// TwinCAT 3 PLC project Mediator
// ProgramVersion: 3.1.4022.2
// libraries:
//   Tc2_Standard, * (Beckhoff Automation GmbH)
//   Tc2_System, * (Beckhoff Automation GmbH)
//   Tc2_Utilities, * (Beckhoff Automation GmbH)
//   Tc3_Module, * (Beckhoff Automation GmbH)
//   VisuSymbols,3.5.10.0,System
// project tree:
//   DUTs/ E_DeliveryStatus.TcDUT, E_MediatorReturnCode.TcDUT, E_MessageList.TcDUT, E_PeerReturnCode.TcDUT, E_PeersList.TcDUT, ST_LinkedListUnit.TcDUT, ST_Mailbox.TcDUT, ST_Message.TcDUT, ST_PeerAccount.TcDUT, E_System.TcDUT, ST_TimeStrings.TcDUT
//   / GlobalTextList.TcGTLO, PlcTask.TcTTO, TL_MessageList.TcTLO, TL_PeersList.TcTLO, Visualisierungsmanager.TcVMO (not stored), VISU_TASK.TcTTO
//   POUs/ CONVEYOR_TEST.TcPOU, MEDIATOR_TEST.TcPOU
//   POUs/System/Components/ FB_Sensor.TcPOU
//   POUs/System/ GTL.TcGVL, GVL_Constants.TcGVL, GVL_System.TcGVL, GVL_SystemParams.TcGVL, I_Module.TcIO, I_Sequence.TcIO
//   POUs/System/LinkedList/ FB_GenericLinkedList.TcPOU, FB_MessageLinkedList.TcPOU, FB_PeerLinkedList.TcPOU
//   POUs/System/Logging/ E_LoggingSeverity.TcDUT, FB_Logging.TcPOU
//   POUs/System/Messaging/ FB_Mediator.TcPOU, FB_Peer.TcPOU, I_Peer.TcIO, F_Message.TcPOU
//   POUs/System/Utilities/Concats/ F_Concat10.TcPOU, F_Concat3.TcPOU, F_Concat4.TcPOU, F_Concat5.TcPOU, F_Concat6.TcPOU, F_Concat7.TcPOU, F_Concat8.TcPOU, F_Concat9.TcPOU
//   POUs/System/Utilities/ FB_WhiteSpaces.TcPOU
//   POUs/TestBlocks/Conveyor/ E_ConveyorPeerSequence.TcDUT, FB_Conveyor.TcPOU, FB_Conveyor1Sequence.TcPOU, FB_Conveyor2Sequence.TcPOU, FB_Conveyor3Sequence.TcPOU, FB_Conveyor4Sequence.TcPOU, FB_ConveyorLogSequence.TcPOU, FB_ConveyorPeerSequence.TcPOU, I_ConveyorSequence.TcIO
//   POUs/TestBlocks/ FB_Void.TcPOU
//   Rezeptur/ RecipeManager.TcRMO (not stored)
//   VISUs/Frames/ Frame_Conveyor.TcVIS, Frame_ConveyorGroup.TcVIS, Frame_ConveyorSmallGroup.TcVIS, Frame_Peer.TcVIS
//   VISUs/ VISU_CONVEYOR_TEST.TcVIS, VISU_MEDIATOR_TEST.TcVIS
// real-time tasks:
//   TASK PlcTask: cycle T#10ms, priority 20, ADS port 350
//   TASK VISU_TASK: cycle T#200000us, priority 30, ADS port 351

CONFIGURATION Mediator
    RESOURCE PLC ON TwinCAT3
        TASK PlcTask(INTERVAL := T#10ms, PRIORITY := 20);
        TASK VISU_TASK(INTERVAL := T#200000us, PRIORITY := 30);
        PROGRAM MEDIATOR_TEST WITH PlcTask : MEDIATOR_TEST;
        PROGRAM VISU_PRG WITH VISU_TASK : VISU_PRG;
    END_RESOURCE
END_CONFIGURATION

// ---- DUTs/E_DeliveryStatus.TcDUT
{attribute 'qualified_only'}
{attribute 'strict'}
TYPE E_DeliveryStatus :
(
	eNO_DELIVERY_INFORMATION := 0,
	eDELIVERY_OK,
	eDELIVERY_REJECTED
)UINT;
END_TYPE

// ---- DUTs/E_MediatorReturnCode.TcDUT
//{attribute 'qualified_only'}
//{attribute 'strict'}
TYPE E_MediatorReturnCode :
(
	eNO_RETURN_CODE := 0,
	ePEER_ALREADY_CONNECTED,
	ePEER_CONNECTED,
	eMAX_NUMBER_OF_CONNECTED_PEERS,
	ePEER_NOT_FOUND,
	eMESSAGE_DISPATCHED,
	eMESSAGE_NOT_DISPATCHED,
	eDISPATCHING_MESSAGE
)UINT;
END_TYPE

// ---- DUTs/E_MessageList.TcDUT
//{attribute 'qualified_only'}
//{attribute 'strict'}
TYPE E_MessageList :
(
	eNO_MESSAGE := 1,
	eCONVEYOR_1_AT_TRANSFER_POINT,
	eCONVEYOR_1_RESUMING_OPERATION,
	eCONVEYOR_2_AT_TRANSFER_POINT,
	eCONVEYOR_2_RESUMING_OPERATION,
	eCONVEYOR_3_AT_TRANSFER_POINT,
	eCONVEYOR_3_RESUMING_OPERATION,
	eCONVEYOR_4_AT_TRANSFER_POINT,
	eCONVEYOR_4_RESUMING_OPERATION,
	eCONVEYOR_1_PACKAGE_DELIVERED,
	eCONVEYOR_2_PACKAGE_DELIVERED,
	eCONVEYOR_3_PACKAGE_DELIVERED,
	eCONVEYOR_4_PACKAGE_DELIVERED
)UINT;
END_TYPE

// ---- DUTs/E_PeerReturnCode.TcDUT
{attribute 'qualified_only'}
{attribute 'strict'}
TYPE E_PeerReturnCode :
(
	eNO_RETURN_CODE := 0,
	eMESSAGE_IN_OUTBOX,
	eMAILBOX_BUSY,
	eMAILBOX_EMPTIED,
	eMAILBOX_EMPTY,
	eNO_NEW_MESSAGE,
	eMATCH_FOUND,
	eNO_MATCH_FOUND
)UINT;
END_TYPE

// ---- DUTs/E_PeersList.TcDUT
//{attribute 'qualified_only'}
//{attribute 'strict'}
TYPE E_PeersList :
(
	ePEER_NO_PEER := 1,
	ePEER_CONVEYOR_1,
	ePEER_CONVEYOR_2,
	ePEER_CONVEYOR_3,
	ePEER_CONVEYOR_4
)UINT;
END_TYPE

// ---- DUTs/ST_LinkedListUnit.TcDUT
TYPE ST_LinkedListUnit :
STRUCT
	
	// 		HEAD <--------------  --------------> TAIL
	//				Previous			Next
	
	pNext : POINTER TO ST_LinkedListUnit;
	pPrevious : POINTER TO ST_LinkedListUnit;
	pVoid : POINTER TO PVOID; // Pointer to the data
	
END_STRUCT
END_TYPE

// ---- DUTs/ST_Mailbox.TcDUT
TYPE ST_Mailbox : 
STRUCT
	stInbox : ST_Message;
	stOutbox : ST_Message;
	bNewMessageAvail : BOOL;
	bSendingMessage : BOOL;
	bMessageSent : BOOL;
END_STRUCT
END_TYPE

// ---- DUTs/ST_Message.TcDUT
{attribute 'enable_dynamic_creation'}
TYPE ST_Message :
STRUCT
	eMessage : E_MessageList;
	eFromPeer : E_PeersList;
	eToPeer : E_PeersList;
	eDeliveryStatus : E_DeliveryStatus;
END_STRUCT
END_TYPE

// ---- DUTs/ST_PeerAccount.TcDUT
TYPE ST_PeerAccount :
STRUCT
	iPeer : I_Peer;
	//fbMessagesList : FB_LinkedListCtrl;
	//nodes : ARRAY[1..nMAX_DATA_ELEMENTS] OF T_LinkedListEntry;
	//hList : T_HLINKEDLIST; //linked list handle
	aMessages : ARRAY[1..nMAX_DATA_ELEMENTS] OF ST_Message;
	nStackPointer : UINT := 1;
	rMailbox : REFERENCE TO ST_MAILBOX; 
	bMailboxFull : BOOL;
	bMailboxEmpty : BOOL := TRUE;
	eDispatchRoutineReturnCode : E_MediatorReturnCode;
END_STRUCT
END_TYPE

// ---- DUTs/E_System.TcDUT
TYPE E_System :
(
	NULL := 0
)UINT;
END_TYPE

// ---- DUTs/ST_TimeStrings.TcDUT
TYPE ST_TimeStrings :
STRUCT
	sYear : STRING;
	sMonth : STRING;
	sDayOfWeek : STRING;
	sDay : STRING;
	sHour : STRING;
	sMinute : STRING;
	sSecond : STRING;
	sMilliseconds : STRING;
END_STRUCT
END_TYPE

// ---- POUs/System/Logging/E_LoggingSeverity.TcDUT
TYPE E_LoggingSeverity :
(
	eNO_LOGGING := 0,
	eINFO,
	eWARNING,
	eDEBUG,
	eERROR,
	eALL
);
END_TYPE

// ---- POUs/TestBlocks/Conveyor/E_ConveyorPeerSequence.TcDUT
{attribute 'qualified_only'}
{attribute 'strict'}
TYPE E_ConveyorPeerSequence :
(
	eIDLE := 0,
	eSTOP,
	eSTART,
	eHOME,
	eWAIT_FOR_ACK,
	eSTOP_AT_SIGNAL,
	eRESUME_OPERATION,
	eEND_SEQUENCE
);
END_TYPE

// ---- POUs/System/GTL.TcGVL
{attribute 'qualified_only'}
VAR_GLOBAL
	gtlPeers : ARRAY[1..nAVAILABLE_PEERS] OF STRING;
	gtlMessages : ARRAY[1..nAVAILABLE_MESSAGES] OF STRING;
	gtlDeliveryStatus : ARRAY[1..nAVAILABLE_DELIVERY_STATUSES] OF STRING;
END_VAR

// ---- POUs/System/GVL_Constants.TcGVL
VAR_GLOBAL CONSTANT
	nMAX_DATA_ELEMENTS : UINT := 4;
	nACTUAL_NUM_PEERS : UINT := 4;
	nMAX_PEER_NUMBER : UINT := 100;
	nMAX_LOG_MESSAGES : UINT := 1000;
	nAVAILABLE_MESSAGES : UINT := 13;
	nAVAILABLE_PEERS : UINT := 5;
	nAVAILABLE_DELIVERY_STATUSES : UINT := 5;
END_VAR

// ---- POUs/System/GVL_System.TcGVL
VAR_GLOBAL
	fbLogList : FB_Logging;
END_VAR

// ---- POUs/System/GVL_SystemParams.TcGVL
{attribute 'qualified_only'}
VAR_GLOBAL CONSTANT
	sLogPath : T_MaxString := '\\Vboxsvr\vm_share\LogFile.csv';//'C:\Users\TC-1\Documents\Log\LogFile.csv';
END_VAR

// ---- POUs/System/I_Module.TcIO
INTERFACE I_Module

PROPERTY AccessModuleName : String
GET
END_GET
SET
END_SET
END_PROPERTY

END_INTERFACE

// ---- POUs/System/I_Sequence.TcIO
INTERFACE I_Sequence

END_INTERFACE

// ---- POUs/System/Messaging/I_Peer.TcIO
INTERFACE I_Peer

METHOD M_GetNextMessage : ST_Message
END_METHOD

METHOD M_GetPeerId : E_PeersList
VAR_INPUT
END_VAR
END_METHOD

METHOD M_IsNewMessageAvailable : BOOL
END_METHOD

METHOD M_RetrieveMailbox : REFERENCE TO ST_MAILBOX
VAR_INPUT
END_VAR
END_METHOD

METHOD M_SendMessage : E_PeerReturnCode
VAR_INPUT
	in_stMessage : ST_Message;
END_VAR
END_METHOD

END_INTERFACE

// ---- POUs/TestBlocks/Conveyor/I_ConveyorSequence.TcIO
INTERFACE I_ConveyorSequence EXTENDS I_Sequence

METHOD M_ConveyorSequence : BOOL
VAR_INPUT
	in_rConveyor : REFERENCE TO FB_Conveyor;
END_VAR
END_METHOD

END_INTERFACE

// ---- POUs/MEDIATOR_TEST.TcPOU
PROGRAM MEDIATOR_TEST
VAR
	fbRecipeManCommands : RecipeManCommands;
	aLogUnits : ARRAY[1..nMAX_LOG_MESSAGES] OF ST_LinkedListUnit;
	aLogMessages :  ARRAY[1..nMAX_LOG_MESSAGES] OF T_MaxString;
	i : INT;

	bTest : BOOL;
	bCloseFile : BOOL; 
//--------------------------------------------------------------------------------------------------------------------------------------------
	fbMediator : FB_Mediator;
	aMediatorInitReturnCodes : ARRAY[1..GVL_Constants.nACTUAL_NUM_PEERS] OF BOOL;
	
	aConveyorPeers : ARRAY[1..GVL_Constants.nACTUAL_NUM_PEERS] OF FB_Conveyor;
	aConveyorPeerSequence : ARRAY[1..GVL_Constants.nACTUAL_NUM_PEERS] OF FB_ConveyorPeerSequence;
	
	fbConveyor1Sequence : FB_Conveyor1Sequence;
	fbConveyor2Sequence : FB_Conveyor2Sequence;
	fbConveyor3Sequence : FB_Conveyor3Sequence;
	fbConveyor4Sequence : FB_Conveyor4Sequence;
	
	rConveyor1 : REFERENCE TO FB_Conveyor;
	rConveyor2 : REFERENCE TO FB_Conveyor;
	rConveyor3 : REFERENCE TO FB_Conveyor;
	rConveyor4 : REFERENCE TO FB_Conveyor;
	
	
	{attribute 'OPC.UA.DA' := '1'}
	bInit : BOOL;
	nMainI : UINT;
	
	(*
	//fbCutPeer : FB_Peer(E_PeersList.ePEER_SCHNEIDEN);
	fbDebugPeer1 : FB_Peer(E_PeersList.ePEER_DEBUG_1);
	fbDebugPeer2 : FB_Peer(E_PeersList.ePEER_DEBUG_2);
	
	eMediatorReturnCode : E_MediatorReturnCode;
	
	bPeer1SendMessage : BOOL;
	bPeer2SendMessage : BOOL;
 	*)
	//DEBUG

	
END_VAR


IF bCloseFile THEN
	bCloseFile := FALSE;
	fbLogList.M_CloseFile();
END_IF

fbMediator();
//fbRecipeManCommands();

IF NOT bInit THEN
	
	fbRecipeManCommands.
		LoadAndWriteRecipe(
			RecipeDefinitionName := 'PeersList',
			RecipeName := 'GTL'
		);
		
	fbMediator.AccessModuleName := 'Mediator';
	rConveyor1 REF= aConveyorPeers[1];
	rConveyor1.M_RegisterSequence(fbConveyor1Sequence);
	rConveyor1.AccessModuleName := GTL.gtlPeers[E_PeersList.ePEER_CONVEYOR_1];
	rConveyor2 REF= aConveyorPeers[2];
	rConveyor2.M_RegisterSequence(fbConveyor2Sequence);
	rConveyor3 REF= aConveyorPeers[3];
	rConveyor3.M_RegisterSequence(fbConveyor3Sequence);
	rConveyor4 REF= aConveyorPeers[4];
	rConveyor4.M_RegisterSequence(fbConveyor4Sequence);
	
	rConveyor1.eSetPeerId := E_PeersList.ePEER_CONVEYOR_1;
	rConveyor2.eSetPeerId := E_PeersList.ePEER_CONVEYOR_2;
	rConveyor3.eSetPeerId := E_PeersList.ePEER_CONVEYOR_3; 
	rConveyor4.eSetPeerId := E_PeersList.ePEER_CONVEYOR_4; 
	
	FOR nMainI := 1 TO GVL_Constants.nACTUAL_NUM_PEERS DO 
		aMediatorInitReturnCodes[nMainI] S= 
			(fbMediator.M_AddPeer(aConveyorPeers[nMainI]) = E_MediatorReturnCode.ePEER_CONNECTED);
		//aConveyorPeers[nMainI].M_RegisterSequence(aConveyorPeerSequence[nMainI]);
		aConveyorPeers[nMainI].in_bSystemStart := TRUE;
	END_FOR	
	
	IF 	aMediatorInitReturnCodes[1]  
		AND aMediatorInitReturnCodes[2]
		AND aMediatorInitReturnCodes[3]
		AND aMediatorInitReturnCodes[4]
		THEN
			bInit := TRUE;
	END_IF
ELSE
	
	FOR nMainI := 1 TO GVL_Constants.nACTUAL_NUM_PEERS DO 
		aConveyorPeers[nMainI]();
	END_FOR	
	
END_IF

END_PROGRAM

// ---- POUs/System/Messaging/FB_Mediator.TcPOU
FUNCTION_BLOCK FB_Mediator IMPLEMENTS I_Module

VAR
	aPeersConnected : ARRAY[1..nMAX_PEER_NUMBER] OF ST_PeerAccount;
	aLogMessages :  ARRAY[1..nMAX_LOG_MESSAGES] OF T_MaxString;
	aPeerUnits : ARRAY[1..nMAX_PEER_NUMBER] OF ST_LinkedListUnit;
	aLogUnits : ARRAY[1..nMAX_LOG_MESSAGES] OF ST_LinkedListUnit;
	
	fbPeersList : FB_PeerLinkedList;
	//fbLogList : FB_Logging;
	
	nStackPointer : UINT := 1;
	bAtLeastOnePeerConnected : BOOL;
	bInit : BOOL;
	i : UINT;
	
	stTestUnit : ST_LinkedListUnit;
	pTestMessage : POINTER TO ST_Message;
	stEmptyMessage : ST_MESSAGE;
	sModuleName : STRING;
	
	//DEBUG:
	//If one of the following variables becomes TRUE, investigation of the cause is mandatory
//--------------------------------------------------------------------------------------------
	bFailedToRelocateToTail : BOOL;
	bNullExceptionWhileDispatching : BOOL;
	bNullExceptionWhileCheckingMailbox : BOOL;
//--------------------------------------------------------------------------------------------


END_VAR
VAR CONSTANT
	
END_VAR

M_Init();
M_CheckMailboxes();
M_DispatchMessages();


PROPERTY AccessModuleName : STRING
GET
AccessModuleName := sModuleName;
END_GET
SET
sModuleName := AccessModuleName;
END_SET
END_PROPERTY

METHOD PUBLIC M_AddPeer : E_MediatorReturnCode
VAR_INPUT
	in_iPeer : I_Peer;
END_VAR
VAR
	i : UINT;
	
END_VAR
IF NOT fbPeersList.bInit THEN
	RETURN;
END_IF

IF nStackPointer > nMAX_PEER_NUMBER THEN
	M_AddPeer := E_MediatorReturnCode.eMAX_NUMBER_OF_CONNECTED_PEERS;
	RETURN;
END_IF

FOR i := 1 TO nMAX_PEER_NUMBER DO
	IF aPeersConnected[i].iPeer = in_iPeer THEN
		M_AddPeer := E_MediatorReturnCode.ePEER_ALREADY_CONNECTED;
		RETURN;	
	END_IF
END_FOR

aPeersConnected[nStackPointer].iPeer := in_iPeer;
aPeersConnected[nStackPointer].rMailbox Ref= in_iPeer.M_RetrieveMailbox();

fbPeersList.M_AddPeerToTail
(
	pPeerToAdd := ADR(aPeersConnected[nStackPointer]),
	pUnitToAdd := ADR(aPeerUnits[nStackPointer])
);

nStackPointer := nStackPointer + 1;

bAtLeastOnePeerConnected := TRUE;

M_AddPeer := E_MediatorReturnCode.ePEER_CONNECTED;
END_METHOD

METHOD PRIVATE M_CheckMailboxes : BOOL

VAR
	nSendersAccount : UINT;
	nSendersStackPointer : UINT;
	stMessageToAdd : ST_Message;
	pPeer : POINTER TO ST_PeerAccount;
END_VAR
IF NOT bAtLeastOnePeerConnected THEN
	RETURN;
END_IF 

FOR nSendersAccount := 1 TO nStackPointer-1 DO
	
(*
	IF nSendersAccount = 1 THEN
		fbPeersList.pGetCurrent := fbPeersList.pHead;
		fbPeersList.nGetNextPosition := 1;
	END_IF
*)

	pPeer :=  fbPeersList.M_GetNextPeer();
	
	IF pPeer = NULL THEN
		//Report null exception
		bNullExceptionWhileCheckingMailbox := TRUE;
		CONTINUE;
	END_IF
	
	IF pPeer^.rMailbox.bMessageSent THEN
		pPeer^.rMailbox.bMessageSent := FALSE;
	END_IF;
	
	//If sender has a message in its outbox, add the message to the list of messages
	//The oldest message always in front of the list (FIFO)
	IF pPeer^.rMailbox.bSendingMessage THEN
		
		nSendersStackPointer := pPeer^.nStackPointer;
		// If the senders account has less then X messages, add the outgoing message to the message list 
		IF nSendersStackPointer <= nMAX_DATA_ELEMENTS THEN
	
			stMessageToAdd := pPeer^.rMailbox.stOutbox;
			
			pPeer^.bMailboxFull := FALSE;
			pPeer^.aMessages[nSendersStackPointer] := stMessageToAdd;		
			pPeer^.nStackPointer := nSendersStackPointer + 1;		
			pPeer^.bMailboxEmpty := FALSE;		
			pPeer^.rMailbox.bSendingMessage := FALSE;
			pPeer^.rMailbox.stOutbox := stEmptyMessage;
	
			//Will be true for only one cycle
			pPeer^.rMailbox.bMessageSent := TRUE;
			
		ELSE
			
			//Mailbox contains more than X messages
			pPeer^.bMailboxFull := TRUE;
			
		END_IF
		
	END_IF
	
END_FOR
END_METHOD

METHOD PRIVATE M_DeleteMessageFromSendersAccount : BOOL
VAR_INPUT
	in_pSenderPeer : POINTER TO ST_PeerAccount;
END_VAR
VAR
	stEmptyMessage : ST_MESSAGE;
	nSendersStackPointer : UINT;
	i : UINT;
END_VAR
IF in_pSenderPeer^.bMailboxEmpty THEN
	RETURN;
END_IF 

nSendersStackPointer := in_pSenderPeer^.nStackPointer;
in_pSenderPeer^.nStackPointer := nSendersStackPointer - 1;

//Only one message was in the list
IF in_pSenderPeer^.nStackPointer = 1 THEN
	
	//Remove oldest message from list
	in_pSenderPeer^.aMessages[1] := stEmptyMessage;
	in_pSenderPeer^.bMailboxEmpty := TRUE;
ELSE
	//Move all the messages by one 
	FOR i := 2 TO nSendersStackPointer-1 DO 
		in_pSenderPeer^.aMessages[i - 1] := 
			in_pSenderPeer^.aMessages[i];
	END_FOR
	
	//Remove newest message from list
	in_pSenderPeer^.aMessages[nSendersStackPointer-1] := stEmptyMessage;
	
END_IF
END_METHOD

METHOD PRIVATE M_DispatchMessages 
VAR_INPUT
END_VAR
VAR_OUTPUT
	
END_VAR
VAR
	nSenderPeer : UINT;
	nReceiverPeer : UINT;
	
	pPeer : POINTER TO ST_PeerAccount;
	pUnit : POINTER TO ST_LinkedListUnit;
	
	nPeerListPosition : UINT;
END_VAR

VAR_INST

END_VAR
IF 	NOT bAtLeastOnePeerConnected 
	OR fbPeersList.M_GetCurrentPosition() = 0
	THEN
	
	RETURN;
END_IF 

FOR nSenderPeer := 1 TO nStackPointer-1 DO
(*	
	IF nSenderPeer = 1 THEN
		fbPeersList.pGetCurrent := fbPeersList.pHead;
		fbPeersList.nGetNextPosition := 1;
	END_IF
*)
	pPeer :=  fbPeersList.M_GetNextPeer();
	
	IF pPeer = NULL THEN
		//Report null exception
		bNullExceptionWhileDispatching := TRUE;
		CONTINUE;
	END_IF
	
	//Check if peer has mail to send
	IF NOT pPeer^.bMailboxEmpty THEN
		
		//Result 0 means peer not found
		nReceiverPeer := M_FindPeer( M_GetReceiverPeerId( pPeer ) );
		
		IF nReceiverPeer > 0 THEN
			
			//Sends the message only when the receiver has emptied its own mailbox
			IF 	NOT aPeersConnected[nReceiverPeer].rMailbox.bNewMessageAvail
				THEN				
				
				M_SendMessage
				(
					in_nReceiverPeer := nReceiverPeer,
					in_pSenderPeer := pPeer 
				);
				
				IF pPeer^.aMessages[1].eDeliveryStatus = E_DeliveryStatus.eDELIVERY_REJECTED THEN
					
					fbLogList.M_Info(
						in_iModule:=THIS^,
						in_sMessage:= 
							F_Concat8(
								'Peer ', 
								GTL.gtlPeers[ pPeer^.iPeer.M_GetPeerId() ],
								' sending message back to Peer ',
								GTL.gtlPeers[ M_GetReceiverPeerId( pPeer ) ],
								': ',
								GTL.gtlMessages[ pPeer^.aMessages[1].eMessage ],
								';Delivery status: ',
								GTL.gtlDeliveryStatus[ pPeer^.aMessages[1].eDeliveryStatus ]						
							) 	
					);
					
				ELSE
					
					fbLogList.M_Info(
						in_iModule:=THIS^,
						in_sMessage:= 
							F_Concat8(
								'Peer ', 
								GTL.gtlPeers[ pPeer^.iPeer.M_GetPeerId() ],
								' sending following message to Peer ',
								GTL.gtlPeers[ M_GetReceiverPeerId( pPeer ) ],
								': ',
								GTL.gtlMessages[ pPeer^.aMessages[1].eMessage ],
								';Delivery status: ',
								GTL.gtlDeliveryStatus[ E_DeliveryStatus.eDELIVERY_OK ]						
							) 	
					);
					
				END_IF

				
				M_DeleteMessageFromSendersAccount(in_pSenderPeer := pPeer);	
							
				pPeer^.eDispatchRoutineReturnCode := eMESSAGE_DISPATCHED;
				
				bFailedToRelocateToTail S= NOT fbPeersList.M_RelocateToTail();


			ELSE
				
				pPeer^.eDispatchRoutineReturnCode := eMESSAGE_NOT_DISPATCHED;
				pPeer^.aMessages[1].eDeliveryStatus := E_DeliveryStatus.eRECEIVERS_MAILBOX_NOT_EMPTY;
				
				fbLogList.M_Info(
					in_iModule:=THIS^,
					in_sMessage:= 
						F_Concat8(
							'Peer ', 
							GTL.gtlPeers[ pPeer^.iPeer.M_GetPeerId() ],
							' failed to send following message to Peer ',
							GTL.gtlPeers[ M_GetReceiverPeerId( pPeer ) ],
							': ',
							GTL.gtlMessages[ pPeer^.aMessages[1].eMessage ],
							';Delivery status: ',
							GTL.gtlDeliveryStatus[ pPeer^.aMessages[1].eDeliveryStatus ]						
						) 	
				);	
				
			END_IF
			
		ELSE
			
			// Report peer not found;	
			
			fbLogList.M_Info(
				in_iModule:=THIS^,
				in_sMessage:= 
					F_Concat8(
						'Peer ', 
						GTL.gtlPeers[ pPeer^.iPeer.M_GetPeerId() ],
						' failed to send following message to Peer ',
						GTL.gtlPeers[ M_GetReceiverPeerId( pPeer ) ],
						': ',
						GTL.gtlMessages[ pPeer^.aMessages[1].eMessage ],
						';Delivery status: ',
						GTL.gtlDeliveryStatus[ E_DeliveryStatus.ePEER_NOT_FOUND ]						
					) 	
			);
			M_DeleteMessageFromSendersAccount(in_pSenderPeer := pPeer);	
			pPeer^.eDispatchRoutineReturnCode := ePEER_NOT_FOUND;
			
		END_IF
				
	END_IF
	
END_FOR
END_METHOD

METHOD PRIVATE M_FindPeer : UINT
VAR_INPUT
	in_ePeer : E_PeersList;
END_VAR
VAR
	i : UINT;
END_VAR
IF 	NOT bAtLeastOnePeerConnected 
	OR in_ePeer = NULL 
	THEN
	
	RETURN;
	
END_IF 

//Check if receiver peer is in the peers list and return position of peer in the list
FOR i := 1 TO nStackPointer - 1 DO
	
	IF aPeersConnected[i].iPeer.M_GetPeerId() = in_ePeer THEN
		
		M_FindPeer := i;
		RETURN;
		
	END_IF
	
END_FOR

M_FindPeer := 0;
END_METHOD

METHOD PRIVATE M_GetReceiverPeerId : E_PeersList
VAR_INPUT
	in_pSenderPeer : POINTER TO ST_PeerAccount;
END_VAR
VAR
	pMessage : POINTER TO ST_Message;
END_VAR
//Extract receivers Id from the oldest message in the list
M_GetReceiverPeerId := in_pSenderPeer^.aMessages[1].eToPeer;
END_METHOD

METHOD PRIVATE M_Init : BOOL
VAR_INPUT
END_VAR
fbPeersList.M_InitLinkedList(aPeerUnits);
fbLogList.M_InitLinkedList(aLogUnits);
fbLogList(in_sPath := GVL_SystemParams.sLogPath);

IF NOT bInit THEN
	bInit := TRUE;
	
	fbLogList.AccessLoggingSeverity := eALL;
	
	FOR i := 1 TO nMAX_LOG_MESSAGES DO
		aLogUnits[i].pVoid := ADR(aLogMessages[i]);
		fbLogList.M_AddToTail(ADR(aLogUnits[i]));
	END_FOR

END_IF
END_METHOD

METHOD PUBLIC M_IsPeerConnected : BOOL
VAR_INPUT
	in_ePeer : E_PeersList;
END_VAR
VAR
	i : UINT;
END_VAR
FOR i := 1 TO nMAX_PEER_NUMBER DO
	
	IF aPeersConnected[i].iPeer.M_GetPeerId() = in_ePeer THEN
		
		M_IsPeerConnected := TRUE;
		RETURN;
		
	END_IF
	
END_FOR
END_METHOD

METHOD PRIVATE M_SendMessage : BOOL
VAR_INPUT
	in_nReceiverPeer : UINT;
	in_pSenderPeer : POINTER TO ST_PeerAccount;
END_VAR
//Dispatch mail after the FIFO principle
aPeersConnected[in_nReceiverPeer].rMailbox.stInbox := in_pSenderPeer^.aMessages[1];
aPeersConnected[in_nReceiverPeer].rMailbox.bNewMessageAvail := TRUE;
END_METHOD

END_FUNCTION_BLOCK

// ---- POUs/System/LinkedList/FB_PeerLinkedList.TcPOU
FUNCTION_BLOCK FB_PeerLinkedList EXTENDS FB_GenericLinkedList
VAR_INPUT
END_VAR
VAR_OUTPUT
END_VAR
VAR
END_VAR

METHOD M_AddPeerToHead : BOOL
VAR_INPUT
	pUnitToAdd : POINTER TO ST_LinkedListUnit;
	pPeerToAdd : POINTER TO ST_PeerAccount;
END_VAR
pUnitToAdd^.pVoid := pPeerToAdd;
SUPER^.M_AddToHead(pUnitToAdd);
END_METHOD

METHOD M_AddPeerToTail : BOOL
VAR_INPUT
	pUnitToAdd : POINTER TO ST_LinkedListUnit;
	pPeerToAdd : POINTER TO ST_PeerAccount;
END_VAR
pUnitToAdd^.pVoid := pPeerToAdd;
SUPER^.M_AddToTail(pUnitToAdd);
END_METHOD

METHOD M_GetHeadPeer : POINTER TO ST_PeerAccount
VAR_INPUT
END_VAR
VAR
	stUnit : POINTER TO ST_LinkedListUnit;
END_VAR
stUnit := SUPER^.M_GetHead();

IF stUnit = NULL THEN
	RETURN;
END_IF

M_GetHeadPeer := stUnit^.pVoid;
END_METHOD

METHOD M_GetNextPeer : POINTER TO ST_PeerAccount
VAR_INPUT
END_VAR
VAR
	stUnit : POINTER TO ST_LinkedListUnit;
END_VAR
stUnit := SUPER^.M_GetNext();

IF stUnit = NULL THEN
	RETURN;
END_IF

M_GetNextPeer := stUnit^.pVoid;
END_METHOD

METHOD M_GetTailPeer : POINTER TO ST_PeerAccount
VAR_INPUT
END_VAR
VAR
	stUnit : POINTER TO ST_LinkedListUnit;
END_VAR
stUnit := SUPER^.M_GetTail();

IF stUnit = NULL THEN
	RETURN;
END_IF

M_GetTailPeer := stUnit^.pVoid;
END_METHOD

END_FUNCTION_BLOCK

// ---- POUs/System/LinkedList/FB_GenericLinkedList.TcPOU
FUNCTION_BLOCK FB_GenericLinkedList
VAR_INPUT
END_VAR
VAR_OUTPUT
	bInit : BOOL;
END_VAR
VAR
	
	pHead : POINTER TO ST_LinkedListUnit;
	pTail : POINTER TO ST_LinkedListUnit;
	pPointer : POINTER TO ST_LinkedListUnit; //Helper
	
	//pGetNext : POINTER TO ST_LinkedListUnit;
	nGetNextPosition : UINT := 1;
	
	pGetCurrent : POINTER TO ST_LinkedListUnit;
	nGetCurrentPosition : UINT := 1;
	
	nSizeOfLinkedList : DINT;
	
	bIsEmpty : BOOL := TRUE;
	bIsFull : BOOL;
	nUnitsInTheList : DINT;
	
		//DEBUG:
	//If one of the following variables becomes TRUE, investigation of the cause is mandatory
//--------------------------------------------------------------------------------------------
	bTriedToRelocatePositionZero : BOOL;
//--------------------------------------------------------------------------------------------
END_VAR

METHOD M_AddToHead : BOOL
VAR_INPUT
	pUnitToAdd : POINTER TO ST_LinkedListUnit;
END_VAR
IF bIsFull THEN
	RETURN;
END_IF

IF bIsEmpty THEN
	pHead := pUnitToAdd;
	pGetCurrent := pHead;
	pTail := pHead;
	pPointer := pHead;
ELSE
	pHead^.pPrevious := pUnitToAdd;
	pUnitToAdd^.pNext := pHead;
	pUnitToAdd^.pPrevious := NULL;
	pHead := pUnitToAdd;	
END_IF

nUnitsInTheList := nUnitsInTheList + 1;
M_CheckUnitsInTheList();

M_AddToHead := TRUE;
END_METHOD

METHOD M_AddToTail : BOOL
VAR_INPUT
	pUnitToAdd : POINTER TO ST_LinkedListUnit;
END_VAR
IF bIsFull THEN
	RETURN;
END_IF

IF bIsEmpty THEN
	pHead := pUnitToAdd;
	pGetCurrent := pHead;
	pTail := pHead;
	pPointer := pHead;
ELSE
	pTail^.pNext := pUnitToAdd;
	pUnitToAdd^.pPrevious := pTail;
	pUnitToAdd^.pNext := NULL;
	pTail := pUnitToAdd;	
END_IF

nUnitsInTheList := nUnitsInTheList + 1;
M_CheckUnitsInTheList();
	
M_AddToTail := TRUE;
END_METHOD

METHOD M_CheckUnitsInTheList : BOOL
VAR_INPUT
END_VAR
IF nUnitsInTheList = nSizeOfLinkedList THEN
	bIsFull := TRUE;
ELSIF nUnitsInTheList < nSizeOfLinkedList THEN
	bIsFull := FALSE;
END_IF

IF nUnitsInTheList > 0 THEN
	bIsEmpty := FALSE;
ELSIF nUnitsInTheList = 0 THEN
	bIsEmpty := TRUE;
END_IF
END_METHOD

METHOD M_FindUnit : BOOL
VAR_INPUT
END_VAR
END_METHOD

METHOD M_GetCurrent : POINTER TO ST_LinkedListUnit
VAR_INPUT
END_VAR
IF bIsEmpty THEN
	RETURN;
END_IF

M_GetCurrent := pGetCurrent;
END_METHOD

METHOD M_GetCurrentPosition : UINT
VAR_INPUT
END_VAR
M_GetCurrentPosition := nGetCurrentPosition;
END_METHOD

METHOD M_GetHead : POINTER TO ST_LinkedListUnit
IF bIsEmpty THEN
	RETURN;
END_IF

M_GetHead := pHead;
END_METHOD

//Gets the next Unit and moves the current pointer forward
METHOD M_GetNext : POINTER TO ST_LinkedListUnit
IF bIsEmpty THEN
	RETURN;
END_IF

//If the search pointer reaches the end, reset the counter and the pointer
IF pGetCurrent = NULL THEN
	pGetCurrent := pHead;
	nGetNextPosition := 1;
	M_GetNext := pGetCurrent;
	//pGetCurrent := pGetCurrent^.pNext;
ELSE
	M_GetNext := pGetCurrent;
	//pGetCurrent := pGetCurrent^.pNext;
END_IF
pGetCurrent := pGetCurrent^.pNext;
nGetCurrentPosition := nGetNextPosition;
//IF nGetCurrentPosition = nUnitsInTheList THEN
//	nGetNextPosition := 1;
//ELSE
	nGetNextPosition := nGetNextPosition + 1;
//END_IF
END_METHOD

METHOD M_GetTail : POINTER TO ST_LinkedListUnit
IF bIsEmpty THEN
	RETURN;
END_IF

M_GetTail := pTail;
END_METHOD

METHOD M_InitLinkedList : BOOL
VAR_IN_OUT
    aLinkedListMemory : ARRAY [*] OF ST_LinkedListUnit;
END_VAR
VAR
	i : DINT;
	nLowerBound : DINT;
	nUpperBound : DINT;
END_VAR
IF bInit THEN
	RETURN;
END_IF

nLowerBound := LOWER_BOUND(aLinkedListMemory,1);
nUpperBound := UPPER_BOUND(aLinkedListMemory,1);

nSizeOfLinkedList := (nUpperBound - nLowerBound) + 1;


bIsEmpty := TRUE;
bInit := TRUE;
M_InitLinkedList := TRUE;
END_METHOD

METHOD M_RelocateHeadToTail : BOOL
VAR
	pUnit : POINTER TO ST_LinkedListUnit;
END_VAR
pUnit := M_RemoveAtLocation(1);

IF pUnit = NULL THEN
	RETURN;
END_IF

//If the current element is the head
//reset counters
(*
IF pUnit = pGetCurrent THEN
	pGetCurrent := pGetCurrent^.pNext;
	nGetNextPosition := 2;
	nGetCurrentPosition := 1;
END_IF
*)
IF M_AddToTail(pUnit) THEN
	M_RelocateHeadToTail := TRUE;
END_IF
END_METHOD

METHOD M_RelocateToHead : BOOL
VAR
	pUnit : POINTER TO ST_LinkedListUnit;
END_VAR
pUnit := M_RemoveAtLocation(M_GetCurrentPosition());

IF pUnit = NULL THEN
	RETURN;
END_IF

IF M_AddToHead(pUnit) THEN
	M_RelocateToHead := TRUE;
END_IF
END_METHOD

METHOD M_RelocateToTail : BOOL
VAR_INPUT
END_VAR
VAR
	pUnit : POINTER TO ST_LinkedListUnit;
END_VAR
pUnit := M_RemoveAtLocation(M_GetCurrentPosition());

IF pUnit = NULL THEN
	RETURN;
END_IF

IF M_AddToTail(pUnit) THEN
	M_RelocateToTail := TRUE;
END_IF
END_METHOD

METHOD M_RemoveAtLocation : POINTER TO ST_LinkedListUnit
VAR_INPUT
	in_nLocation : UINT;
END_VAR
VAR
	nCounter : UINT;
END_VAR
IF 	bIsEmpty 
	OR in_nLocation > nUnitsInTheList
	OR in_nLocation = 0
	THEN
	
	IF  in_nLocation = 0 
		AND NOT bIsEmpty 
		THEN
		
		bTriedToRelocatePositionZero := TRUE;
	END_IF
	
	RETURN;
END_IF

pPointer := pHead;
IF in_nLocation = 1 THEN
	M_RemoveAtLocation := M_RemoveHead();
	RETURN;
ELSIF in_nLocation = nUnitsInTheList THEN
	M_RemoveAtLocation := M_RemoveTail();
	RETURN;
ELSE
	
	FOR nCounter := 2 TO in_nLocation DO
		pPointer := pPointer^.pNext;
	END_FOR

END_IF

M_RemoveAtLocation := pPointer;

nUnitsInTheList := nUnitsInTheList - 1;
M_CheckUnitsInTheList();

pPointer := pPointer^.pPrevious;
pPointer^.pNext := pPointer^.pNext^.pNext;
pPointer := pPointer^.pNext;
pPointer^.pPrevious := pPointer^.pPrevious^.pPrevious;
END_METHOD

METHOD M_RemoveHead : POINTER TO ST_LinkedListUnit
VAR_INPUT
END_VAR
IF bIsEmpty THEN
	RETURN;
END_IF

M_RemoveHead := pHead;

IF nUnitsInTheList = 1 THEN
	nUnitsInTheList := 0;
	bIsEmpty := TRUE;	
	pHead := NULL;
	pTail := NULL;
	pPointer := NULL;
ELSE
	pHead := pHead^.pNext;
	pHead^.pPrevious := NULL; 	
	nUnitsInTheList := nUnitsInTheList - 1;
END_IF

M_CheckUnitsInTheList();
END_METHOD

METHOD M_RemoveTail : POINTER TO ST_LinkedListUnit
VAR_INPUT
END_VAR
IF bIsEmpty THEN
	RETURN;
END_IF

M_RemoveTail := pTail;

IF nUnitsInTheList = 1 THEN
	nUnitsInTheList := 0;
	bIsEmpty := TRUE;	
	pHead := NULL;
	pTail := NULL;
	pPointer := NULL;
ELSE
	pTail := pTail^.pPrevious;
	pTail^.pNext := NULL; 	
	nUnitsInTheList := nUnitsInTheList - 1;
END_IF

M_CheckUnitsInTheList();
END_METHOD

END_FUNCTION_BLOCK

// ---- POUs/System/Utilities/Concats/F_Concat8.TcPOU
FUNCTION F_Concat8 : STRING(255)
VAR_INPUT
	String1 : STRING(255);
	String2 : STRING(255);
	String3 : STRING(255);
	String4 : STRING(255);
	String5 : STRING(255);
	String6 : STRING(255);
	String7 : STRING(255);
	String8 : STRING(255);
END_VAR
VAR
END_VAR

F_Concat8 := F_Concat7(String2,String3,String4,String5,String6,String7,String8);
F_Concat8 := CONCAT(String1,F_Concat8);

END_FUNCTION

// ---- POUs/System/Utilities/Concats/F_Concat7.TcPOU
FUNCTION F_Concat7 : STRING(255)
VAR_INPUT
	String1 : STRING(255);
	String2 : STRING(255);
	String3 : STRING(255);
	String4 : STRING(255);
	String5 : STRING(255);
	String6 : STRING(255);
	String7 : STRING(255);
END_VAR
VAR
END_VAR

F_Concat7 := F_Concat6(String2,String3,String4,String5,String6,String7);
F_Concat7 := CONCAT(String1,F_Concat7);

END_FUNCTION

// ---- POUs/System/Utilities/Concats/F_Concat6.TcPOU
FUNCTION F_Concat6 : STRING(255)
VAR_INPUT
	String1 : STRING(255);
	String2 : STRING(255);
	String3 : STRING(255);
	String4 : STRING(255);
	String5 : STRING(255);
	String6 : STRING(255);
END_VAR
VAR
END_VAR

F_Concat6 := F_Concat5(String2,String3,String4,String5,String6);
F_Concat6 := CONCAT(String1,F_Concat6);

END_FUNCTION

// ---- POUs/System/Utilities/Concats/F_Concat5.TcPOU
FUNCTION F_Concat5 : STRING(255)
VAR_INPUT
	String1 : STRING(255);
	String2 : STRING(255);
	String3 : STRING(255);
	String4 : STRING(255);
	String5 : STRING(255);
END_VAR
VAR
END_VAR

F_Concat5 := F_Concat4(String2,String3,String4,String5);
F_Concat5 := CONCAT(String1,F_Concat5);

END_FUNCTION

// ---- POUs/System/Utilities/Concats/F_Concat4.TcPOU
FUNCTION F_Concat4 : STRING(255)
VAR_INPUT
	String1 : STRING(255);
	String2 : STRING(255);
	String3 : STRING(255);
	String4 : STRING(255);
END_VAR
VAR
END_VAR

F_Concat4 := F_CONCAT3(String2,String3,String4);
F_Concat4 := CONCAT(String1,F_Concat4);

END_FUNCTION

// ---- POUs/System/Utilities/Concats/F_Concat3.TcPOU
FUNCTION F_Concat3 : STRING(255)
VAR_INPUT
	String1 : STRING(255);
	String2 : STRING(255);
	String3 : STRING(255);
END_VAR
VAR
END_VAR

F_Concat3 := CONCAT(String1,CONCAT(String2,String3));

END_FUNCTION

// ---- POUs/TestBlocks/Conveyor/FB_Conveyor.TcPOU
FUNCTION_BLOCK FB_Conveyor EXTENDS FB_Peer IMPLEMENTS I_Module
VAR_INPUT
	in_bSystemStart : BOOL;
	in_bStop : BOOL;
	in_bStart : BOOL;
END_VAR
VAR_OUTPUT
	out_fbSensorStop : FB_Sensor;
	out_fbSensorMaterialDispatch : FB_Sensor;
	out_fbSensorSignal : FB_Sensor;
END_VAR
VAR	
	{attribute 'OPC.UA.DA' := '1'}
	bStartMotor AT%Q* : BOOL;
	iSequence : I_ConveyorSequence;
	sModuleName : STRING;
END_VAR

M_CallComponents();
IF in_bSystemStart THEN
	M_RunSequence();
END_IF

PROPERTY AccessModuleName : STRING
GET
AccessModuleName := sModuleName;
END_GET
SET
sModuleName := AccessModuleName;
END_SET
END_PROPERTY

METHOD M_CallComponents : E_PeerReturnCode
VAR_INPUT
END_VAR
out_fbSensorSignal();
out_fbSensorMaterialDispatch();
out_fbSensorStop();
END_METHOD

METHOD M_RegisterSequence : BOOL
VAR_INPUT
	in_iSequence : I_ConveyorSequence;
END_VAR
iSequence := in_iSequence;
END_METHOD

METHOD M_RunSequence : BOOL
VAR_INPUT
END_VAR
IF iSequence = NULL THEN
	RETURN;
END_IF

iSequence.M_ConveyorSequence(this^);
END_METHOD

METHOD M_StartConveyor : BOOL
VAR_INPUT
END_VAR
bStartMotor := TRUE;
END_METHOD

METHOD M_StopConveyor : E_PeerReturnCode
VAR_INPUT
END_VAR
bStartMotor := FALSE;
END_METHOD

END_FUNCTION_BLOCK

// ---- POUs/System/Messaging/FB_Peer.TcPOU
FUNCTION_BLOCK FB_Peer IMPLEMENTS I_Peer
VAR_INPUT
END_VAR
VAR_OUTPUT
END_VAR
VAR
	ePeer : E_PeersList;
	stMailbox : ST_Mailbox; 
END_VAR

PROPERTY eSetPeerId : E_PeersList
SET
ePeer := eSetPeerId;
END_SET
END_PROPERTY

METHOD M_CompareMessage : E_PeerReturnCode
VAR_INPUT
	in_stMessage : ST_Message;
END_VAR
VAR
	stIncomingMessage : ST_MESSAGE;
END_VAR
IF M_IsNewMessageAvailable() THEN
	
	stIncomingMessage := M_GetNextMessage();
	IF 	stIncomingMessage.eMessage = in_stMessage.eMessage
		AND stIncomingMessage.eFromPeer = in_stMessage.eFromPeer
		THEN
		
		M_CompareMessage := E_PeerReturnCode.eMATCH_FOUND;
		
	ELSE
		
		M_CompareMessage := E_PeerReturnCode.eNO_MATCH_FOUND;
	
	END_IF
	
ELSE

	M_CompareMessage := E_PeerReturnCode.eNO_NEW_MESSAGE;	
	
END_IF
END_METHOD

METHOD M_CompareMessageAndEmptyMailbox : E_PeerReturnCode
VAR_INPUT
	in_stMessage : ST_Message;
END_VAR
VAR
	stMessage : ST_Message;
	eTmpEval : E_PeerReturnCode;
END_VAR
M_CompareMessageAndEmptyMailbox := M_CompareMessage(in_stMessage);

IF M_CompareMessageAndEmptyMailbox = E_PeerReturnCode.eNO_MATCH_FOUND THEN
	stMessage := M_GetNextMessage();
	stMessage.eDeliveryStatus := E_DeliveryStatus.eDELIVERY_REJECTED;
	stMessage.eToPeer := stMessage.eFromPeer;
	stMessage.eFromPeer := M_GetPeerId();
	eTmpEval := M_SendMessage(stMessage);
END_IF

IF eTmpEval = E_PeerReturnCode.eMESSAGE_IN_OUTBOX
	OR M_CompareMessageAndEmptyMailbox = E_PeerReturnCode.eMATCH_FOUND
	THEN
	
	M_EmptyMailbox();
	
END_IF
END_METHOD

METHOD M_EmptyMailbox : E_PeerReturnCode
VAR_INPUT
END_VAR
VAR
	stEmptyMessage : ST_MESSAGE;
END_VAR
IF M_IsNewMessageAvailable() THEN
	stMailbox.stInbox := stEmptyMessage;
	stMailbox.bNewMessageAvail := FALSE;
	M_EmptyMailbox := E_PeerReturnCode.eMAILBOX_EMPTIED;
ELSE
	M_EmptyMailbox := E_PeerReturnCode.eMAILBOX_EMPTY;
END_IF
END_METHOD

METHOD M_GetNextMessage : ST_Message
IF M_IsNewMessageAvailable() THEN
	M_GetNextMessage := stMailbox.stInbox;
END_IF
END_METHOD

METHOD M_GetPeerId : E_PeersList
M_GetPeerId := ePeer;
END_METHOD

METHOD M_IsNewMessageAvailable : BOOL
M_IsNewMessageAvailable := stMailbox.bNewMessageAvail;
END_METHOD

METHOD M_RetrieveMailbox : REFERENCE TO ST_MAILBOX
VAR_INPUT
END_VAR
M_RetrieveMailbox Ref= stMailbox;
END_METHOD

METHOD M_SendMessage : E_PeerReturnCode
VAR_INPUT
	in_stMessage : ST_Message;
END_VAR
IF NOT stMailbox.bSendingMessage THEN
	stMailbox.stOutbox := in_stMessage;
	stMailbox.bSendingMessage := TRUE;
	M_SendMessage := E_PeerReturnCode.eMESSAGE_IN_OUTBOX;
ELSE
	M_SendMessage := E_PeerReturnCode.eMAILBOX_BUSY;
END_IF
END_METHOD

END_FUNCTION_BLOCK

// ---- POUs/System/Components/FB_Sensor.TcPOU
FUNCTION_BLOCK FB_Sensor
VAR_INPUT
END_VAR
VAR_OUTPUT
END_VAR
VAR
	{attribute 'OPC.UA.DA' := '1'}
	bSignal  AT%I* : BOOL;	
	fbRTrig : R_TRIG;
END_VAR

fbRTrig(CLK:= bSignal, Q=> );

PROPERTY GetSignal : BOOL
GET
GetSignal := bSignal;
END_GET
END_PROPERTY

PROPERTY GetTriggerSignal : BOOL
GET
GetTriggerSignal := fbRTrig.Q;
END_GET
END_PROPERTY

END_FUNCTION_BLOCK

// ---- POUs/TestBlocks/Conveyor/FB_ConveyorPeerSequence.TcPOU
FUNCTION_BLOCK FB_ConveyorPeerSequence IMPLEMENTS I_ConveyorSequence
VAR_INPUT

END_VAR
VAR_OUTPUT
END_VAR
VAR
	nStep : E_ConveyorPeerSequence;
END_VAR

METHOD M_ConveyorAction : BOOL
VAR_INPUT
	in_stFirstMessage : ST_Message;
	in_stMessageToWaitFor : ST_Message;
	in_stSecondMessage : ST_Message;
	in_rConveyor : REFERENCE TO FB_Conveyor;
END_VAR
VAR_INST
	nConveyorActionStep : UINT;
END_VAR
CASE nConveyorActionStep OF
	
	0:
		IF 	in_rConveyor.M_SendMessage
			(	
				in_stFirstMessage
			) 
			= E_PeerReturnCode.eMESSAGE_IN_OUTBOX 
			THEN
			
			nConveyorActionStep := 10;
			
		END_IF
		
	10:
		
	
		IF 	in_rConveyor.M_CompareMessageAndEmptyMailbox
			(	
				in_stMessageToWaitFor
			) 
			= E_PeerReturnCode.eMATCH_FOUND 
			THEN
			
			nConveyorActionStep := 20;
			
		END_IF

	20:
		
		IF 	in_rConveyor.M_SendMessage
			(	
				in_stSecondMessage
			) 
			= E_PeerReturnCode.eMESSAGE_IN_OUTBOX 
			THEN
			
			nConveyorActionStep := 0;
			M_ConveyorAction := TRUE;
			
		END_IF
		
END_CASE
END_METHOD


METHOD M_ConveyorSequence : BOOL
VAR_INPUT
	in_rConveyor : REFERENCE TO FB_Conveyor;
END_VAR
CASE nStep OF
	
	E_ConveyorPeerSequence.eIDLE:
	
		IF in_rConveyor.in_bStart THEN
			nStep := E_ConveyorPeerSequence.eSTART;
		END_IF
				
	E_ConveyorPeerSequence.eSTART:
		
		in_rConveyor.M_StartConveyor();
		nStep := E_ConveyorPeerSequence.eSTOP_AT_SIGNAL;

	E_ConveyorPeerSequence.eSTOP_AT_SIGNAL:
	
		IF in_rConveyor.out_fbSensorStop.GetTriggerSignal THEN
			in_rConveyor.M_StopConveyor();
			nStep := E_ConveyorPeerSequence.eWAIT_FOR_ACK;
		END_IF
	
	E_ConveyorPeerSequence.eWAIT_FOR_ACK:
		
		IF M_SubjectiveAction(in_rConveyor) THEN
			nStep := E_ConveyorPeerSequence.eRESUME_OPERATION;
		END_IF
	
	E_ConveyorPeerSequence.eRESUME_OPERATION:
		
		in_rConveyor.M_StartConveyor();
		IF in_rConveyor.out_fbSensorMaterialDispatch.GetTriggerSignal THEN
			in_rConveyor.M_StopConveyor();
			nStep := E_ConveyorPeerSequence.eEND_SEQUENCE;
		END_IF
	
	E_ConveyorPeerSequence.eEND_SEQUENCE:
		
END_CASE
END_METHOD

METHOD M_SubjectiveAction : BOOL
VAR_INPUT
	in_rConveyor : REFERENCE TO FB_Conveyor;
END_VAR

VAR
	stFirstMessageToSend : ST_Message;
	stMessageToWaitFor : ST_Message;
	stSecondMessageToSend : ST_Message;
END_VAR
CASE in_rConveyor.M_GetPeerId() OF

	E_PeersList.ePEER_CONVEYOR_1:
	
		stFirstMessageToSend :=
			F_Message(
				eFromPeer := ePEER_CONVEYOR_1,
				eToPeer := ePEER_CONVEYOR_2,
				eMessage := eCONVEYOR_1_AT_TRANSFER_POINT
			);
			
		stMessageToWaitFor := 
			F_Message(
				eFromPeer := ePEER_CONVEYOR_4,
				eToPeer := ePEER_CONVEYOR_1,
				eMessage := eCONVEYOR_4_AT_TRANSFER_POINT
			);
			
		stSecondMessageToSend := 
			F_Message(
				eFromPeer := ePEER_CONVEYOR_1,
				eToPeer := ePEER_CONVEYOR_2,
				eMessage := eCONVEYOR_1_RESUMING_OPERATION
			);
			
	E_PeersList.ePEER_CONVEYOR_2:
		
		stFirstMessageToSend :=
			F_Message(
				eFromPeer := ePEER_CONVEYOR_2,
				eToPeer := ePEER_CONVEYOR_3,
				eMessage := eCONVEYOR_2_AT_TRANSFER_POINT
			);
			
		stMessageToWaitFor := 
			F_Message(
				eFromPeer := ePEER_CONVEYOR_1,
				eToPeer := ePEER_CONVEYOR_2,
				eMessage := eCONVEYOR_1_RESUMING_OPERATION
			);
			
		stSecondMessageToSend := 
			F_Message(
				eFromPeer := ePEER_CONVEYOR_2,
				eToPeer := ePEER_CONVEYOR_3,
				eMessage := eCONVEYOR_2_RESUMING_OPERATION
			);	
	
	E_PeersList.ePEER_CONVEYOR_3:
	
		stFirstMessageToSend :=
			F_Message(
				eFromPeer := ePEER_CONVEYOR_3,
				eToPeer := ePEER_CONVEYOR_4,
				eMessage := eCONVEYOR_3_AT_TRANSFER_POINT
			);
			
		stMessageToWaitFor := 
			F_Message(
				eFromPeer := ePEER_CONVEYOR_2,
				eToPeer := ePEER_CONVEYOR_3,
				eMessage := eCONVEYOR_2_RESUMING_OPERATION
			);
			
		stSecondMessageToSend := 
			F_Message(
				eFromPeer := ePEER_CONVEYOR_3,
				eToPeer := ePEER_CONVEYOR_4,
				eMessage := eCONVEYOR_3_RESUMING_OPERATION
			);
	
	E_PeersList.ePEER_CONVEYOR_4:
	
		stFirstMessageToSend :=
			F_Message(
				eFromPeer := ePEER_CONVEYOR_4,
				eToPeer := ePEER_CONVEYOR_1,
				eMessage := eCONVEYOR_4_AT_TRANSFER_POINT
			);
			
		stMessageToWaitFor := 
			F_Message(
				eFromPeer := ePEER_CONVEYOR_3,
				eToPeer := ePEER_CONVEYOR_4,
				eMessage := eCONVEYOR_3_RESUMING_OPERATION
			);
			
		stSecondMessageToSend := 
			F_Message(
				eFromPeer := ePEER_CONVEYOR_4,
				eToPeer := ePEER_NO_PEER,
				eMessage := eNO_MESSAGE
			);	

END_CASE

M_SubjectiveAction := 
	M_ConveyorAction(
		in_rConveyor := in_rConveyor,
		in_stFirstMessage := stFirstMessageToSend,
		in_stMessageToWaitFor := stMessageToWaitFor,
		in_stSecondMessage := stSecondMessageToSend
	);
END_METHOD

END_FUNCTION_BLOCK

// ---- POUs/System/Messaging/F_Message.TcPOU
FUNCTION F_Message : ST_Message
VAR_INPUT
	eMessage : E_MessageList;
	eFromPeer : E_PeersList;
	eToPeer : E_PeersList;
END_VAR
VAR
END_VAR

F_Message.eMessage := eMessage;
F_Message.eFromPeer := eFromPeer;
F_Message.eToPeer := eToPeer;

END_FUNCTION

// ---- POUs/TestBlocks/Conveyor/FB_Conveyor1Sequence.TcPOU
FUNCTION_BLOCK FB_Conveyor1Sequence IMPLEMENTS I_ConveyorSequence
VAR_INPUT
END_VAR
VAR_OUTPUT
END_VAR
VAR
	nStep : UINT;
END_VAR


METHOD M_ConveyorSequence : BOOL
VAR_INPUT
	in_rConveyor	: REFERENCE TO FB_Conveyor;
END_VAR
VAR
	stMessage : ST_Message;
	ePeerReturnCode : E_PeerReturnCode;
END_VAR
CASE nStep OF
	
	0 :
 
		IF in_rConveyor.in_bStart THEN
			in_rConveyor.M_StartConveyor();
			nStep := 20;
		END_IF
		
	20 :
	
		IF in_rConveyor.out_fbSensorStop.GetTriggerSignal THEN
			in_rConveyor.M_StopConveyor();
			nStep := 30;
		END_IF
		
	30 :
	
		stMessage :=
			F_Message(
				eFromPeer := E_PeersList.ePEER_CONVEYOR_1,
				eToPeer := E_PeersList.ePEER_CONVEYOR_2,
				eMessage := E_MessageList.eCONVEYOR_1_AT_TRANSFER_POINT
			);
		in_rConveyor.M_SendMessage(stMessage);
 		nStep := 40;
	
	40 : 
	
		stMessage := 
			F_Message(
				eFromPeer := E_PeersList.ePEER_CONVEYOR_4,
				eToPeer := E_PeersList.ePEER_CONVEYOR_1,
				eMessage := E_MessageList.eCONVEYOR_4_AT_TRANSFER_POINT
			);
			
		ePeerReturnCode := in_rConveyor.M_CompareMessageAndEmptyMailbox(stMessage);
		
		IF ePeerReturnCode = E_PeerReturnCode.eMATCH_FOUND THEN
			in_rConveyor.M_StartConveyor();
			nStep := 50;
		END_IF
	
	50: 
			
		IF in_rConveyor.out_fbSensorMaterialDispatch.GetTriggerSignal THEN
			stMessage := 
				F_Message(
					eFromPeer := E_PeersList.ePEER_CONVEYOR_1,
					eToPeer := E_PeersList.ePEER_CONVEYOR_2,
					eMessage := E_MessageList.eCONVEYOR_1_PACKAGE_DELIVERED
				);
			in_rConveyor.M_StopConveyor();
			in_rConveyor.M_SendMessage(stMessage);
			nStep := 0;
		END_IF		
				
END_CASE
END_METHOD

END_FUNCTION_BLOCK

// ---- POUs/TestBlocks/Conveyor/FB_Conveyor2Sequence.TcPOU
FUNCTION_BLOCK FB_Conveyor2Sequence IMPLEMENTS I_ConveyorSequence
VAR_INPUT
END_VAR
VAR_OUTPUT
END_VAR
VAR
	nStep : UINT;
END_VAR


METHOD M_ConveyorSequence : BOOL
VAR_INPUT
	in_rConveyor	: REFERENCE TO FB_Conveyor;
END_VAR
VAR
	stMessage : ST_Message;
	ePeerReturnCode : E_PeerReturnCode;
END_VAR
CASE nStep OF
	
	0 :
 
		stMessage := 
			F_Message(
				eFromPeer := E_PeersList.ePEER_CONVEYOR_1,
				eToPeer := E_PeersList.ePEER_CONVEYOR_2,
				eMessage := E_MessageList.eCONVEYOR_1_AT_TRANSFER_POINT
			);
			
		ePeerReturnCode := in_rConveyor.M_CompareMessageAndEmptyMailbox(stMessage);
		
		IF ePeerReturnCode = E_PeerReturnCode.eMATCH_FOUND THEN
			in_rConveyor.M_StartConveyor();
			nStep := 20;
		END_IF
		
	20 :
	
		IF in_rConveyor.out_fbSensorStop.GetTriggerSignal THEN
			in_rConveyor.M_StopConveyor();
			nStep := 30;
		END_IF
		
	30 :
	
		stMessage :=
			F_Message(
				eFromPeer := E_PeersList.ePEER_CONVEYOR_2,
				eToPeer := E_PeersList.ePEER_CONVEYOR_3,
				eMessage := E_MessageList.eCONVEYOR_2_AT_TRANSFER_POINT
			);
			
		in_rConveyor.M_SendMessage(stMessage);
 		nStep := 40;
	
	40 : 
	
		stMessage := 
			F_Message(
				eFromPeer := E_PeersList.ePEER_CONVEYOR_1,
				eToPeer := E_PeersList.ePEER_CONVEYOR_2,
				eMessage := E_MessageList.eCONVEYOR_1_PACKAGE_DELIVERED
			);
			
		ePeerReturnCode := in_rConveyor.M_CompareMessageAndEmptyMailbox(stMessage);
		
		IF ePeerReturnCode = E_PeerReturnCode.eMATCH_FOUND THEN
			in_rConveyor.M_StartConveyor();
			nStep := 50;
		END_IF
	
	50: 
			
		IF in_rConveyor.out_fbSensorMaterialDispatch.GetTriggerSignal THEN
			
			stMessage := 
				F_Message(
					eFromPeer := E_PeersList.ePEER_CONVEYOR_2,
					eToPeer := E_PeersList.ePEER_CONVEYOR_3,
					eMessage := E_MessageList.eCONVEYOR_2_PACKAGE_DELIVERED
				);
				
			in_rConveyor.M_StopConveyor();
			in_rConveyor.M_SendMessage(stMessage);
			nStep := 0;
			
		END_IF		
				
END_CASE
END_METHOD

END_FUNCTION_BLOCK

// ---- POUs/TestBlocks/Conveyor/FB_Conveyor3Sequence.TcPOU
FUNCTION_BLOCK FB_Conveyor3Sequence IMPLEMENTS I_ConveyorSequence
VAR_INPUT
END_VAR
VAR_OUTPUT
END_VAR
VAR
	nStep : UINT;
END_VAR


METHOD M_ConveyorSequence : BOOL
VAR_INPUT
	in_rConveyor	: REFERENCE TO FB_Conveyor;
END_VAR
VAR
	stMessage : ST_Message;
	ePeerReturnCode : E_PeerReturnCode;
END_VAR
CASE nStep OF
	
	0 :
 
		stMessage := 
			F_Message(
				eFromPeer := E_PeersList.ePEER_CONVEYOR_2,
				eToPeer := E_PeersList.ePEER_CONVEYOR_3,
				eMessage := E_MessageList.eCONVEYOR_2_AT_TRANSFER_POINT
			);
			
		ePeerReturnCode := in_rConveyor.M_CompareMessageAndEmptyMailbox(stMessage);
		
		IF ePeerReturnCode = E_PeerReturnCode.eMATCH_FOUND THEN
			in_rConveyor.M_StartConveyor();
			nStep := 20;
		END_IF
		
	20 :
	
		IF in_rConveyor.out_fbSensorStop.GetTriggerSignal THEN
			in_rConveyor.M_StopConveyor();
			nStep := 30;
		END_IF
		
	30 :
	
		stMessage :=
			F_Message(
				eFromPeer := E_PeersList.ePEER_CONVEYOR_3,
				eToPeer := E_PeersList.ePEER_CONVEYOR_4,
				eMessage := E_MessageList.eCONVEYOR_3_AT_TRANSFER_POINT
			);
			
		in_rConveyor.M_SendMessage(stMessage);
 		nStep := 40;
	
	40 : 
	
		stMessage := 
			F_Message(
				eFromPeer := E_PeersList.ePEER_CONVEYOR_2,
				eToPeer := E_PeersList.ePEER_CONVEYOR_3,
				eMessage := E_MessageList.eCONVEYOR_2_PACKAGE_DELIVERED
			);
			
		ePeerReturnCode := in_rConveyor.M_CompareMessageAndEmptyMailbox(stMessage);
		
		IF ePeerReturnCode = E_PeerReturnCode.eMATCH_FOUND THEN
			in_rConveyor.M_StartConveyor();
			nStep := 50;
		END_IF
	
	50: 
			
		IF in_rConveyor.out_fbSensorMaterialDispatch.GetTriggerSignal THEN
			
			stMessage := 
				F_Message(
					eFromPeer := E_PeersList.ePEER_CONVEYOR_3,
					eToPeer := E_PeersList.ePEER_CONVEYOR_4,
					eMessage := E_MessageList.eCONVEYOR_3_PACKAGE_DELIVERED
				);
				
			in_rConveyor.M_StopConveyor();
			in_rConveyor.M_SendMessage(stMessage);
			nStep := 0;
			
		END_IF		
				
END_CASE
END_METHOD

END_FUNCTION_BLOCK

// ---- POUs/TestBlocks/Conveyor/FB_Conveyor4Sequence.TcPOU
FUNCTION_BLOCK FB_Conveyor4Sequence IMPLEMENTS I_ConveyorSequence
VAR_INPUT
END_VAR
VAR_OUTPUT
END_VAR
VAR
	nStep : UINT;
END_VAR


METHOD M_ConveyorSequence : BOOL
VAR_INPUT
	in_rConveyor	: REFERENCE TO FB_Conveyor;
END_VAR
VAR
	stMessage : ST_Message;
	ePeerReturnCode : E_PeerReturnCode;
END_VAR
CASE nStep OF
	
	0 :
 
		stMessage := 
			F_Message(
				eFromPeer := E_PeersList.ePEER_CONVEYOR_3,
				eToPeer := E_PeersList.ePEER_CONVEYOR_4,
				eMessage := E_MessageList.eCONVEYOR_3_AT_TRANSFER_POINT
			);
			
		ePeerReturnCode := in_rConveyor.M_CompareMessageAndEmptyMailbox(stMessage);
		
		IF ePeerReturnCode = E_PeerReturnCode.eMATCH_FOUND THEN
			in_rConveyor.M_StartConveyor();
			nStep := 20;
		END_IF
		
	20 :
	
		IF in_rConveyor.out_fbSensorStop.GetTriggerSignal THEN
			in_rConveyor.M_StopConveyor();
			nStep := 30;
		END_IF
		
	30 :
	
		stMessage :=
			F_Message(
				eFromPeer := E_PeersList.ePEER_CONVEYOR_4,
				eToPeer := E_PeersList.ePEER_CONVEYOR_1,
				eMessage := E_MessageList.eCONVEYOR_4_AT_TRANSFER_POINT
			);
			
		in_rConveyor.M_SendMessage(stMessage);
 		nStep := 40;
	
	40 : 
	
		stMessage := 
			F_Message(
				eFromPeer := E_PeersList.ePEER_CONVEYOR_3,
				eToPeer := E_PeersList.ePEER_CONVEYOR_4,
				eMessage := E_MessageList.eCONVEYOR_3_PACKAGE_DELIVERED
			);
			
		ePeerReturnCode := in_rConveyor.M_CompareMessageAndEmptyMailbox(stMessage);
		
		IF ePeerReturnCode = E_PeerReturnCode.eMATCH_FOUND THEN
			in_rConveyor.M_StartConveyor();
			nStep := 50;
		END_IF
	
	50: 
			
		IF in_rConveyor.out_fbSensorMaterialDispatch.GetTriggerSignal THEN
			
			stMessage := 
				F_Message(
					eFromPeer := E_PeersList.ePEER_CONVEYOR_4,
					eToPeer := E_PeersList.ePEER_NO_PEER,
					eMessage := E_MessageList.eNO_MESSAGE
				);
				
			in_rConveyor.M_StopConveyor();
			in_rConveyor.M_SendMessage(stMessage);
			nStep := 0;
			
		END_IF		
				
END_CASE
END_METHOD

END_FUNCTION_BLOCK

// ---- POUs/System/Logging/FB_Logging.TcPOU
FUNCTION_BLOCK FB_Logging EXTENDS FB_GenericLinkedList
VAR_INPUT
	in_sPath : T_MaxString;
END_VAR
VAR_OUTPUT
END_VAR
VAR
	
	fbFileOpen : FB_FileOpen;
	fbFileWrite : FB_FileWrite;
	fbFileClose : FB_FileClose;
	
	fbSystemTime : NT_GetTime;
	stTime : TIMESTRUCT;
	stTimeStrings : ST_TimeStrings;
	sTimeString : STRING;
	nLenghtOfTimeString : INT;
	nWriteSize : UINT;
	fbWhiteSpaces : FB_WhiteSpaces;
	
	bLogInit : BOOL;
	nInitStep : UINT;
	
	aTmpBuffer : ARRAY[1..nMAX_LOG_MESSAGES] OF T_MaxString;
	aByteBuffer : ARRAY[1..nMAX_LOG_MESSAGES*256] OF BYTE;
	aZeroByteBuffer : ARRAY[1..nMAX_LOG_MESSAGES*256] OF BYTE;
	nByteBufferSP : UINT := 1;
	
	nEntriesToWrite : UINT;
	bLogOverflow : BOOL;
	bOverflowSignaled : BOOL;
	nLinesOverflow : UINT;
	
	eCurrentLoggingSeverity : E_LoggingSeverity;
	
	fbGetCurTaskIdx  : GETCURTASKINDEX;
    nCycleCount      : UDINT;
	
END_VAR
VAR CONSTANT
	sLogOverflow : T_MAXSTRING := 'Log overflow detected:';
END_VAR

M_Cyclic();
M_CheckOverflow();

IF M_Init() THEN
	M_WriteToFile();
END_IF

PROPERTY AccessLoggingSeverity : E_LoggingSeverity
GET
AccessLoggingSeverity := eCurrentLoggingSeverity;
END_GET
SET
eCurrentLoggingSeverity := AccessLoggingSeverity;
END_SET
END_PROPERTY

METHOD M_AddMessageToHead : BOOL
VAR_INPUT
	pUnitToAdd : POINTER TO ST_LinkedListUnit;
	pMessageToAdd : POINTER TO T_MaxString;
END_VAR
pUnitToAdd^.pVoid := pMessageToAdd;
SUPER^.M_AddToHead(pUnitToAdd);
END_METHOD

METHOD M_AddMessageToTail : BOOL
VAR_INPUT
	pUnitToAdd : POINTER TO ST_LinkedListUnit;
	pMessageToAdd : POINTER TO T_MaxString;
END_VAR
pUnitToAdd^.pVoid := pMessageToAdd;
SUPER^.M_AddToTail(pUnitToAdd);
END_METHOD

METHOD M_CheckOverflow : BOOL
VAR_INPUT
END_VAR
IF bLogOverflow THEN
	
	bLogOverflow := FALSE;
	
 	ADSLOGDINT(
		msgCtrlMask := ADSLOG_MSGTYPE_ERROR,
		msgFmtStr := CONCAT(sLogOverflow,' %d lines.'),		
		dintArg := nLinesOverflow
	);
	
END_IF
END_METHOD

METHOD M_CloseFile : BOOL
VAR_INPUT
END_VAR
fbFileClose(bExecute := TRUE);
fbFileClose.bExecute := FALSE;
END_METHOD

METHOD M_Cyclic : BOOL
VAR_INPUT
END_VAR
fbGetCurTaskIdx();
nCycleCount := _TaskInfo[fbGetCurTaskIdx.index].CycleCount;

fbSystemTime(
	NETID:= , 
	START:= NOT fbSystemTime.start, 
	TMOUT:= , 
	BUSY=> , 
	ERR=> , 
	ERRID=> , 
	TIMESTR=> stTime);

M_FormatTimeToString();	

fbFileOpen(
	sNetId:= , 
	sPathName:= in_sPath, 
	nMode:= FOPEN_MODEAPPEND OR FOPEN_MODETEXT, 
	ePath:= , 
	bExecute:= , 
	tTimeout:= , 
	bBusy=> , 
	bError=> , 
	nErrId=> , 
	hFile=> fbFileWrite.hFile);
	
fbFileWrite(
	sNetId:= , 
	hFile:= , 
	pWriteBuff:=, 
	cbWriteLen:= , 
	bExecute:= FALSE, 
	tTimeout:= , 
	bBusy=> , 
	bError=> , 
	nErrId=> , 
	cbWrite=> 
);

fbFileClose(
	sNetId:= , 
	hFile:= fbFileOpen.hFile, 
	bExecute:= , 
	tTimeout:= , 
	bBusy=> , 
	bError=> , 
	nErrId=> );
END_METHOD

METHOD M_Debug : BOOL
VAR_INPUT
	in_sMessage : T_MaxString;
	in_iModule : I_Module;
END_VAR
VAR
	stUnit : POINTER TO ST_LinkedListUnit;
	pMessage : POINTER TO T_MaxString;
END_VAR
IF 	NOT M_SeverityCheck(eDEBUG)
	OR in_iModule = NULL
 	THEN
		
	RETURN;
	
END_IF

nEntriesToWrite := nEntriesToWrite + 1;

IF nEntriesToWrite > nMAX_LOG_MESSAGES THEN
	RETURN;
END_IF

stUnit := M_GetNext();
pMessage := stUnit^.pVoid;

pMessage^ := F_Concat4( 'DEBUG:;' , in_iModule.AccessModuleName ,';', in_sMessage);
END_METHOD

METHOD M_Error : BOOL
VAR_INPUT
	in_sMessage : T_MaxString;
	in_iModule : I_Module;
END_VAR
VAR
	stUnit : POINTER TO ST_LinkedListUnit;
	pMessage : POINTER TO T_MaxString;
END_VAR
IF 	NOT M_SeverityCheck(eERROR)
	OR in_iModule = NULL
 	THEN
		
	RETURN;
	
END_IF

nEntriesToWrite := nEntriesToWrite + 1;

IF nEntriesToWrite > nMAX_LOG_MESSAGES THEN
	RETURN;
END_IF

stUnit := M_GetNext();
pMessage := stUnit^.pVoid;

pMessage^ := F_Concat4( 'ERROR:;' , in_iModule.AccessModuleName ,';', in_sMessage);
END_METHOD

METHOD M_FormatTimeToString 
VAR_INPUT
END_VAR
stTimeStrings.sYear := WORD_TO_STRING(stTime.wYear);
stTimeStrings.sMonth := WORD_TO_STRING(stTime.wMonth);
stTimeStrings.sDayOfWeek := WORD_TO_STRING(stTime.wDayOfWeek);
stTimeStrings.sDay := WORD_TO_STRING(stTime.wDay);
stTimeStrings.sHour := WORD_TO_STRING(stTime.wHour);
stTimeStrings.sMinute := WORD_TO_STRING(stTime.wMinute);
stTimeStrings.sSecond := WORD_TO_STRING(stTime.wSecond);
stTimeStrings.sMilliseconds := WORD_TO_STRING(stTime.wMilliseconds);

sTimeString := 
	F_Concat10(
		stTimeStrings.sYear,
		'.',
		stTimeStrings.sMonth,
		'.',
		stTimeStrings.sDay,
		' | ',
		stTimeStrings.sHour,
		':',
		stTimeStrings.sMinute,
		':'
	);
	
sTimeString := 
	F_Concat4(
		sTimeString,
		stTimeStrings.sSecond,
		':',
		stTimeStrings.sMilliseconds
	);
	
nLenghtOfTimeString := LEN(sTimeString);
END_METHOD

METHOD M_GetHeadMessage : POINTER TO T_MaxString
VAR_INPUT
END_VAR
VAR
	stUnit : POINTER TO ST_LinkedListUnit;
END_VAR
stUnit := SUPER^.M_GetHead();

IF stUnit = NULL THEN
	RETURN;
END_IF

M_GetHeadMessage := stUnit^.pVoid;
END_METHOD

METHOD M_GetNextMessage : POINTER TO T_MaxString
VAR
	stUnit : POINTER TO ST_LinkedListUnit;
END_VAR
stUnit := SUPER^.M_GetNext();

IF stUnit = NULL THEN
	RETURN;
END_IF

M_GetNextMessage := stUnit^.pVoid;
END_METHOD

METHOD M_GetTailMessage : POINTER TO T_MaxString
VAR_INPUT
END_VAR
VAR
	stUnit : POINTER TO ST_LinkedListUnit;
END_VAR
stUnit := SUPER^.M_GetTail();

IF stUnit = NULL THEN
	RETURN;
END_IF

M_GetTailMessage := stUnit^.pVoid;
END_METHOD

METHOD M_Info : BOOL
VAR_INPUT
	in_sMessage : T_MaxString;
	in_iModule : I_Module;
END_VAR
VAR
	stUnit : POINTER TO ST_LinkedListUnit;
	pMessage : POINTER TO T_MaxString;
END_VAR
IF 	NOT M_SeverityCheck(eINFO)
	OR in_iModule = NULL
 	THEN
		
	RETURN;
	
END_IF

nEntriesToWrite := nEntriesToWrite + 1;

IF nEntriesToWrite > nMAX_LOG_MESSAGES THEN
	RETURN;
END_IF

stUnit := M_GetNext();
pMessage := stUnit^.pVoid;

pMessage^ := F_Concat4( 'INFO:;' , in_iModule.AccessModuleName ,';', in_sMessage);
END_METHOD

METHOD M_Init : BOOL
VAR_INPUT
END_VAR
VAR
	i : UINT;
END_VAR
CASE nInitStep OF
	
	0: 
		fbFileOpen.bExecute := TRUE;
		nInitStep := 20;
		
	20:
		IF NOT fbFileOpen.bBusy THEN
			nInitStep := 30;
		END_IF
		
	30: 
		bLogInit := TRUE;
		M_Init := TRUE;
		
END_CASE
END_METHOD

METHOD M_Log : BOOL
VAR_INPUT
	in_sMessage : T_MaxString;
END_VAR
VAR
	stUnit : POINTER TO ST_LinkedListUnit;
	pMessage : POINTER TO T_MaxString;
END_VAR
nEntriesToWrite := nEntriesToWrite + 1;

IF nEntriesToWrite > nMAX_LOG_MESSAGES THEN
	RETURN;
END_IF

stUnit := M_GetNext();
pMessage := stUnit^.pVoid;

pMessage^ := in_sMessage;
END_METHOD

METHOD M_SeverityCheck : BOOL
VAR_INPUT
	eCallerSeverity : E_LoggingSeverity;
END_VAR
M_SeverityCheck := (eCurrentLoggingSeverity=eCallerSeverity) OR (eCurrentLoggingSeverity=eALL);
END_METHOD

METHOD M_Warning : BOOL
VAR_INPUT
	in_sMessage : T_MaxString;
	in_iModule : I_Module;
END_VAR
VAR
	stUnit : POINTER TO ST_LinkedListUnit;
	pMessage : POINTER TO T_MaxString;
END_VAR
IF 	NOT M_SeverityCheck(eWARNING)
	OR in_iModule = NULL
 	THEN
		
	RETURN;
	
END_IF

nEntriesToWrite := nEntriesToWrite + 1;

IF nEntriesToWrite > nMAX_LOG_MESSAGES THEN
	RETURN;
END_IF

stUnit := M_GetNext();
pMessage := stUnit^.pVoid;

pMessage^ := F_Concat4( 'WARNING:;' , in_iModule.AccessModuleName ,';', in_sMessage);
END_METHOD

METHOD M_WriteToFile : BOOL
VAR_INPUT
END_VAR
VAR
	i : UINT;
	j : UINT;
	pBuffer : POINTER TO T_MaxString;
	nSizeOfString : INT;
	nSizeToFill : INT;
	sFillString : STRING;
	
END_VAR
//Check how many lines have been logged
IF nEntriesToWrite > nMAX_LOG_MESSAGES THEN
	nLinesOverflow := nEntriesToWrite - nMAX_LOG_MESSAGES;
	nEntriesToWrite := nMAX_LOG_MESSAGES;
	bLogOverflow := TRUE;
END_IF

IF 	NOT fbFileWrite.bBusy 
	AND nEntriesToWrite > 0 
	AND nEntriesToWrite <= nMAX_LOG_MESSAGES 
	THEN

	MEMCPY(ADR(aByteBuffer),ADR(aZeroByteBuffer),SIZEOF(aZeroByteBuffer));
	//Use LEN to calculate the size of the string
	FOR i := 1 TO nEntriesToWrite DO
		
		pBuffer := M_GetHead()^.pVoid;
		
		aTmpBuffer[i] := F_Concat6(pBuffer^,';',sTimeString,';',UDINT_TO_STRING(nCycleCount),'$N');
		
		MEMCPY(ADR(aByteBuffer[nByteBufferSP]),ADR(aTmpBuffer[i]),LEN(aTmpBuffer[i]));
		nByteBufferSP := nByteBufferSP + INT_TO_UINT(LEN(aTmpBuffer[i]));

		M_RelocateHeadToTail();
		
	END_FOR
	
	fbFileWrite(
		bExecute:= TRUE,
		pWriteBuff := ADR(aByteBuffer),
		cbWriteLen := nByteBufferSP
	);
	
	nEntriesToWrite := 0;
	nByteBufferSP := 1;
	
END_IF
END_METHOD

END_FUNCTION_BLOCK

// ---- POUs/System/Utilities/FB_WhiteSpaces.TcPOU
FUNCTION_BLOCK FB_WhiteSpaces
VAR_INPUT
END_VAR
VAR_OUTPUT
	sWhiteSpace : T_MaxString;
END_VAR
VAR
	bInit : BOOL;
	i : UINT;

END_VAR

IF NOT bInit THEN
	bInit := TRUE;
	FOR i := 1 TO SIZEOF(T_MAXSTRING) DO
		sWhiteSpace := Concat(sWhiteSpace,' ');
	END_FOR
END_IF

END_FUNCTION_BLOCK

// ---- POUs/System/Utilities/Concats/F_Concat10.TcPOU
FUNCTION F_Concat10 : STRING(255)
VAR_INPUT
	String1 : STRING(255);
	String2 : STRING(255);
	String3 : STRING(255);
	String4 : STRING(255);
	String5 : STRING(255);
	String6 : STRING(255);
	String7 : STRING(255);
	String8 : STRING(255);
	String9 : STRING(255);
	String10 : STRING(255);
END_VAR
VAR
END_VAR

F_Concat10 := F_Concat9(String2,String3,String4,String5,String6,String7,String8,String9,String10);
F_Concat10 := CONCAT(String1,F_Concat10);

END_FUNCTION

// ---- POUs/System/Utilities/Concats/F_Concat9.TcPOU
FUNCTION F_Concat9 : STRING(255)
VAR_INPUT
	String1 : STRING(255);
	String2 : STRING(255);
	String3 : STRING(255);
	String4 : STRING(255);
	String5 : STRING(255);
	String6 : STRING(255);
	String7 : STRING(255);
	String8 : STRING(255);
	String9 : STRING(255);
END_VAR
VAR
END_VAR

F_Concat9 := F_Concat8(String2,String3,String4,String5,String6,String7,String8,String9);
F_Concat9 := CONCAT(String1,F_Concat9);

END_FUNCTION

// ---- POUs/CONVEYOR_TEST.TcPOU
PROGRAM CONVEYOR_TEST
VAR
	bInit : BOOL;
	bCloseFile : BOOL;
	
	i : INT;
	aLogUnits : ARRAY[1..nMAX_LOG_MESSAGES] OF ST_LinkedListUnit;
	aLogMessages :  ARRAY[1..nMAX_LOG_MESSAGES] OF T_MaxString;
	
	aConveyors : ARRAY[1..8] OF FB_Conveyor;
	aSequences : ARRAY[1..8] OF FB_ConveyorLogSequence;
	
END_VAR

fbLogList.M_InitLinkedList(aLogUnits);
fbLogList(in_sPath := GVL_SystemParams.sLogPath);

IF NOT bInit THEN
	bInit := TRUE;
	
	fbLogList.AccessLoggingSeverity := eALL;
	
	FOR i := 1 TO nMAX_LOG_MESSAGES DO
		aLogUnits[i].pVoid := ADR(aLogMessages[i]);
		fbLogList.M_AddToTail(ADR(aLogUnits[i]));
	END_FOR
	
	FOR i := 1 TO 8 DO
		aConveyors[i].AccessModuleName := CONCAT('Modul ', INT_TO_STRING(i));
		aConveyors[i].M_RegisterSequence(aSequences[i]);
		aConveyors[i].in_bSystemStart := TRUE;
	END_FOR
END_IF

FOR i := 1 TO 8 DO
	aConveyors[i]();
END_FOR

IF bCloseFile THEN
	bCloseFile := FALSE;
	fbLogList.M_CloseFile();
END_IF

END_PROGRAM

// ---- POUs/TestBlocks/Conveyor/FB_ConveyorLogSequence.TcPOU
FUNCTION_BLOCK FB_ConveyorLogSequence IMPLEMENTS I_ConveyorSequence
VAR_INPUT
END_VAR
VAR_OUTPUT
END_VAR
VAR
	nStep : UINT;
END_VAR


METHOD M_ConveyorSequence : BOOL
VAR_INPUT
	in_rConveyor	: REFERENCE TO FB_Conveyor;
END_VAR
CASE nStep OF
	0: 
		IF in_rConveyor.in_bStart THEN
			in_rConveyor.in_bStart := FALSE;
			in_rConveyor.M_StartConveyor();
			nStep := 10;
		END_IF
		
	10: 
		IF in_rConveyor.out_fbSensorSignal.GetTriggerSignal THEN
			fbLogList.M_Warning(
				in_iModule:=in_rConveyor,
				in_sMessage:='Material erfasst!'	
			);
		END_IF
		
		IF in_rConveyor.in_bStop THEN
			in_rConveyor.in_bStop := FALSE;
			in_rConveyor.M_StopConveyor();
			nStep := 20;
		END_IF
 
	20:
		
		nStep := 30;
	
	30:
	
END_CASE
END_METHOD

END_FUNCTION_BLOCK

// ---- POUs/System/LinkedList/FB_MessageLinkedList.TcPOU
FUNCTION_BLOCK FB_MessageLinkedList EXTENDS FB_GenericLinkedList
VAR_INPUT
END_VAR
VAR_OUTPUT
END_VAR
VAR
END_VAR

METHOD M_AddMessageToHead : BOOL
VAR_INPUT
	pUnitToAdd : POINTER TO ST_LinkedListUnit;
	pMessageToAdd : POINTER TO ST_Message;
END_VAR
pUnitToAdd^.pVoid := pMessageToAdd;
SUPER^.M_AddToHead(pUnitToAdd);
END_METHOD

METHOD M_AddMessageToTail : BOOL
VAR_INPUT
	pUnitToAdd : POINTER TO ST_LinkedListUnit;
	pMessageToAdd : POINTER TO ST_Message;
END_VAR
pUnitToAdd^.pVoid := pMessageToAdd;
SUPER^.M_AddToTail(pUnitToAdd);
END_METHOD

METHOD M_GetHeadMessage : POINTER TO ST_Message
VAR_INPUT
END_VAR
VAR
	stUnit : POINTER TO ST_LinkedListUnit;
END_VAR
stUnit := SUPER^.M_GetHead();

IF stUnit = NULL THEN
	RETURN;
END_IF

M_GetHeadMessage := stUnit^.pVoid;
END_METHOD

METHOD M_GetNextMessage : POINTER TO ST_Message
VAR
	stUnit : POINTER TO ST_LinkedListUnit;
END_VAR
stUnit := SUPER^.M_GetNext();

IF stUnit = NULL THEN
	RETURN;
END_IF

M_GetNextMessage := stUnit^.pVoid;
END_METHOD

METHOD M_GetTailMessage : POINTER TO ST_Message
VAR_INPUT
END_VAR
VAR
	stUnit : POINTER TO ST_LinkedListUnit;

END_VAR
stUnit := SUPER^.M_GetTail();

IF stUnit = NULL THEN
	RETURN;
END_IF

M_GetTailMessage := stUnit^.pVoid;
END_METHOD

END_FUNCTION_BLOCK

// ---- POUs/TestBlocks/FB_Void.TcPOU
FUNCTION_BLOCK FB_Void
VAR_INPUT
END_VAR
VAR_OUTPUT
END_VAR
VAR
	pSequenceMaster : POINTER TO PVOID;
	fbConveyor : FB_Conveyor;
	fbVoidConveyor : FB_Conveyor;
	pConveyor : POINTER TO FB_Conveyor;
END_VAR

pSequenceMaster := ADR(fbConveyor);

pConveyor := pSequenceMaster;

END_FUNCTION_BLOCK

// ---- GlobalTextList.TcGTLO
TEXTLIST GlobalTextList
  677 = '%'
  256 = '%s'
  306 = 'Close Logfile'
  649 = 'Conveyor 1'
  572 = 'Conveyor 2'
  789 = 'Conveyor 3'
  508 = 'Conveyor 4'
  429 = 'Conveyor Group'
  921 = 'Conveyor group'
  377 = 'Conveyor Small Group'
  82 = 'Conveyor small group'
  875 = 'Delivery Status'
  774 = 'DeliveryStatus'
  824 = 'Head'
  965 = 'Inbox'
  526 = 'Mailbox empty'
  175 = 'Mailbox Empty'
  245 = 'Mailbox full'
  962 = 'Mailbox Full'
  431 = 'MAIN.fbMediator.aPeersConnected[INDEX].bMailboxEmpty'
  706 = 'Message'
  630 = 'Message sent'
  281 = 'New message avail'
  324 = 'Nodes'
  652 = 'Outbox'
  184 = 'Peer'
  749 = 'Peer 1 send message to Peer 2'
  330 = 'Peer 2 send message to Peer 1'
  629 = 'Sending message'
  58 = 'Sensor 1'
  499 = 'Sensor 2'
  859 = 'Sensor 3'
  285 = 'Sensor 4'
  724 = 'Stack Pointer'
  10 = 'Start'
  126 = 'Stop'
  818 = 'Tail'
END_TEXTLIST

// ---- TL_MessageList.TcTLO
TEXTLIST TL_MessageList
  7 = 'eCONVEYOR_1_AT_TRANSFER_POINT'
  8 = 'eCONVEYOR_1_RESUMING_OPERATION'
  9 = 'eCONVEYOR_2_AT_TRANSFER_POINT'
  10 = 'eCONVEYOR_2_RESUMING_OPERATION'
  11 = 'eCONVEYOR_3_AT_TRANSFER_POINT'
  12 = 'eCONVEYOR_3_RESUMING_OPERATION'
  13 = 'eCONVEYOR_4_AT_TRANSFER_POINT'
  14 = 'eCONVEYOR_4_RESUMING_OPERATION'
  15 = ''
  16 = ''
  17 = ''
   = ''
END_TEXTLIST

// ---- TL_PeersList.TcTLO
TEXTLIST TL_PeersList
  0 = 'No peer'
  1 = 'Debug 1'
  2 = 'Debug 2'
  3 = 'Schneiden'
  4 = 'Umlenkung'
  5 = 'Bereitstellung'
  6 = 'Conveyor 1'
  7 = 'Conveyor 2'
  8 = 'Conveyor 3'
  9 = 'Conveyor 4'
  10 = 'Conveyor 5'
   = ''
END_TEXTLIST

// ---- VISUs/Frames/Frame_Conveyor.TcVIS
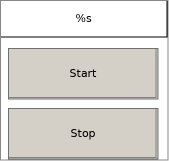
VISUALIZATION Frame_Conveyor  // 169x161
VAR_IN_OUT
	vio_fbConveyor : FB_Conveyor;
END_VAR
    Group (0,0 167x159)
        Button (8,48 150x51), "Start"
            tap vio_fbConveyor.in_bStart
        Button (8,108 150x51), "Stop"
            tap vio_fbConveyor.in_bStop
        Rectangle (0,0 167x37), "%s", text variable: vio_fbConveyor.sModuleName
END_VISUALIZATION

// ---- VISUs/Frames/Frame_ConveyorGroup.TcVIS
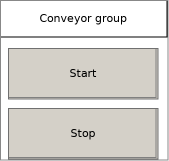
VISUALIZATION Frame_ConveyorGroup  // 169x161
VAR_IN_OUT
	vio_fbConveyor1 : FB_Conveyor;
	vio_fbConveyor2 : FB_Conveyor;
	vio_fbConveyor3 : FB_Conveyor;
	vio_fbConveyor4 : FB_Conveyor;
	vio_fbConveyor5 : FB_Conveyor;
	vio_fbConveyor6 : FB_Conveyor;
	vio_fbConveyor7 : FB_Conveyor;
	vio_fbConveyor8 : FB_Conveyor;
END_VAR
    Button (8,48 150x51), "Start"
        OnMouseDown: execute {
            vio_fbConveyor1.in_bStart := TRUE;
            vio_fbConveyor2.in_bStart := TRUE;
            vio_fbConveyor3.in_bStart := TRUE;
            vio_fbConveyor4.in_bStart := TRUE;
            vio_fbConveyor5.in_bStart := TRUE;
            vio_fbConveyor6.in_bStart := TRUE;
            vio_fbConveyor7.in_bStart := TRUE;
            vio_fbConveyor8.in_bStart := TRUE;
        }
    Button (8,108 150x51), "Stop"
        OnMouseDown: execute {
            vio_fbConveyor1.in_bStop := TRUE;
            vio_fbConveyor2.in_bStop := TRUE;
            vio_fbConveyor3.in_bStop := TRUE;
            vio_fbConveyor4.in_bStop := TRUE;
            vio_fbConveyor5.in_bStop := TRUE;
            vio_fbConveyor6.in_bStop := TRUE;
            vio_fbConveyor7.in_bStop := TRUE;
            vio_fbConveyor8.in_bStop := TRUE;
        }
    Rectangle (0,0 167x37), "Conveyor group"
END_VISUALIZATION

// ---- VISUs/Frames/Frame_ConveyorSmallGroup.TcVIS
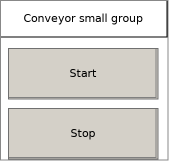
VISUALIZATION Frame_ConveyorSmallGroup  // 169x161
VAR_IN_OUT
	vio_fbConveyor1 : FB_Conveyor;
	vio_fbConveyor2 : FB_Conveyor;
	vio_fbConveyor3 : FB_Conveyor;
	vio_fbConveyor4 : FB_Conveyor;
END_VAR
    Button (8,48 150x51), "Start"
        OnMouseDown: execute {
            vio_fbConveyor1.in_bStart := TRUE;
            vio_fbConveyor2.in_bStart := TRUE;
            vio_fbConveyor3.in_bStart := TRUE;
            vio_fbConveyor4.in_bStart := TRUE;
        }
    Button (8,108 150x51), "Stop"
        OnMouseDown: execute {
            vio_fbConveyor1.in_bStop := TRUE;
            vio_fbConveyor2.in_bStop := TRUE;
            vio_fbConveyor3.in_bStop := TRUE;
            vio_fbConveyor4.in_bStop := TRUE;
        }
    Rectangle (0,0 167x37), "Conveyor small group"
END_VISUALIZATION

// ---- VISUs/Frames/Frame_Peer.TcVIS
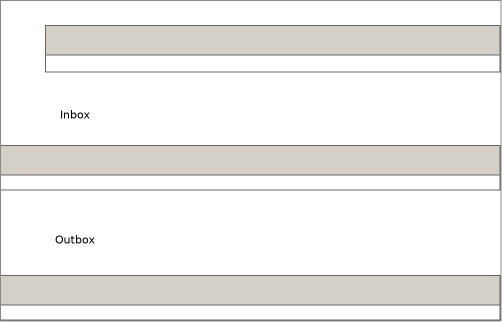
VISUALIZATION Frame_Peer  // 502x322
VAR_IN_OUT
	vio_fbPeer : FB_Peer;
	vio_stMailbox : ST_MAILBOX;
END_VAR
    Table (45,25 455x47), data array: vio_fbPeer.stMailbox
        p3854506369: vio_fbPeer.stMailbox.stInbox
        p1892666644: vio_fbPeer.stMailbox.stOutbox
        p338671338: vio_fbPeer.stMailbox.bNewMessageAvail
        p2170511999: vio_fbPeer.stMailbox.bSendingMessage
        p3723444502: vio_fbPeer.stMailbox.bMessageSent
        p1218418051: vio_fbPeer.stMailbox.eMessage
        p746581629: vio_fbPeer.stMailbox.ePeer
        p3104783080: vio_fbPeer.stMailbox.eDeliveryStatus
        p1755163831: New message avail
        p4092479075: Sending message
        p2237128397: Message sent
    Table (0,275 500x45), data array: vio_stMailbox.stOutbox
        p3854506369: vio_stMailbox.stOutbox.eMessage
        p1892666644: vio_stMailbox.stOutbox.ePeer
        p2170511999: vio_stMailbox.bSendingMessage
        p3723444502: vio_stMailbox.bMessageSent
        p338671338: vio_stMailbox.stOutbox.eDeliveryStatus
        p1755163831: Delivery Status
    Label (0,100 150x30), "Inbox"
    Label (0,225 150x30), "Outbox"
    Table (0,145 500x45), data array: vio_stMailbox.stInbox
        p3854506369: vio_stMailbox.stInbox.eMessage
        p1892666644: vio_stMailbox.stInbox.ePeer
        p2170511999: vio_stMailbox.bSendingMessage
        p3723444502: vio_stMailbox.bMessageSent
        p338671338: vio_stMailbox.stInbox.eDeliveryStatus
        p1755163831: Delivery Status
END_VISUALIZATION

// ---- VISUs/VISU_CONVEYOR_TEST.TcVIS
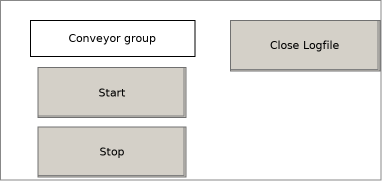
VISUALIZATION VISU_CONVEYOR_TEST  // 382x181
    Frame (30,20 167x159)
        shows Frame_ConveyorGroup(vio_fbConveyor1 := CONVEYOR_TEST.aConveyors[1], vio_fbConveyor2 := CONVEYOR_TEST.aConveyors[2], vio_fbConveyor3 := CONVEYOR_TEST.aConveyors[3], vio_fbConveyor4 := CONVEYOR_TEST.aConveyors[4], vio_fbConveyor5 := CONVEYOR_TEST.aConveyors[5], vio_fbConveyor6 := CONVEYOR_TEST.aConveyors[6], vio_fbConveyor7 := CONVEYOR_TEST.aConveyors[7], vio_fbConveyor8 := CONVEYOR_TEST.aConveyors[8])
    Button (230,20 150x51), "Close Logfile"
        tap CONVEYOR_TEST.bCloseFile
END_VISUALIZATION

// ---- VISUs/VISU_MEDIATOR_TEST.TcVIS
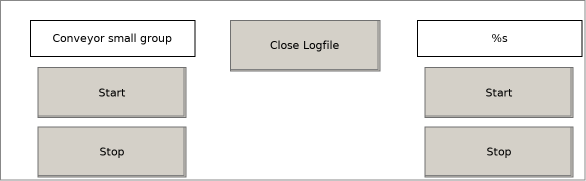
VISUALIZATION VISU_MEDIATOR_TEST  // 586x181
    Frame (30,20 167x159)
        shows Frame_ConveyorSmallGroup(vio_fbConveyor1 := MEDIATOR_TEST.aConveyorPeers[1], vio_fbConveyor2 := MEDIATOR_TEST.aConveyorPeers[2], vio_fbConveyor3 := MEDIATOR_TEST.aConveyorPeers[3], vio_fbConveyor4 := MEDIATOR_TEST.aConveyorPeers[4])
    Button (230,20 150x51), "Close Logfile"
        tap MEDIATOR_TEST.bCloseFile
    Frame (417,20 167x159)
        shows Frame_Conveyor(vio_fbConveyor := MEDIATOR_TEST.aConveyorPeers[1])
END_VISUALIZATION
